# B&R Automation Studio project NAELD004C00R10L518F00 (part 18)

#### Act_OptP1030Save.st
```iecst
ACTION Act_OptP1030Save:

	CASE p_tyNtParamCurr.eProjMag OF
		LDMagDual, LDMagTriple:
			IF tyP1030MagSet.tyMagSet.tyBtnSave.bRtCompl = TRUE THEN
				IF usiSaveMagRcpStep = 0 THEN
					//Mask Table
					tyP1030MagSet.tyMagSet.tyTableRecipe.uiMaskRtStat				:= FALSE;
					tyP1030MagSet.tyMagSet.tyBtnDelete.uiMaskRtStat					:= FALSE;

					p_tyC0008MsgBox ACCESS ADR(tyP1030MagSet.tyMsgBoxSaveAsk);

					IF tyP1030MagSet.tyMsgBoxSaveAsk.tyBtnYes.bRtCompl = TRUE THEN
						tyP1030MagSet.tyMsgBoxSaveAsk.tyBtnYes.bRtCompl				:= FALSE;
						tyP1030MagSet.tyMsgBoxSaveAsk.tyBtnYes.bValue				:= FALSE;

						p_tyC0008MsgBox ACCESS ADR(tyP1030MagSet.tyMsgBoxHide);

						usiSaveMagRcpStep	:= 1;

					ELSIF tyP1030MagSet.tyMsgBoxSaveAsk.tyBtnNo.bRtCompl = TRUE THEN
						tyP1030MagSet.tyMsgBoxSaveAsk.tyBtnNo.bRtCompl				:= FALSE;
						tyP1030MagSet.tyMsgBoxSaveAsk.tyBtnNo.bValue				:= FALSE;

						p_tyC0008MsgBox ACCESS ADR(tyP1030MagSet.tyMsgBoxHide);

						usiSaveMagRcpStep	:= 99;

					END_IF

				ELSIF usiSaveMagRcpStep = 1 THEN
					tyMagRcpInfoIn.sRcpNm					:= tyP1030MagSet.tyMagSet.tyStringRecipeNm.sValue;
					tyMagRcpInfoIn.diSltToSltInUM			:= tyP1030MagSet.tyMagSet.tyNumSltToSltDist.diValue;
					tyMagRcpInfoIn.diTtlSlt					:= tyP1030MagSet.tyMagSet.tyNumMaxSlt.diValue;
					tyMagRcpInfoIn.diMag1Slt1PosInUM		:= tyP1030MagSet.tyMagSet.tyNumLifterMag1Slt1Pos.diValue;
					tyMagRcpInfoIn.diMag2Slt1PosInUM		:= tyP1030MagSet.tyMagSet.tyNumLifterMag2Slt1Pos.diValue;
					tyMagRcpInfoIn.diMag3Slt1PosInUM		:= tyP1030MagSet.tyMagSet.tyNumLifterMag3Slt1Pos.diValue;
					tyMagRcpInfoIn.diMag4Slt1PosInUM		:= tyP1030MagSet.tyMagSet.tyNumLifterMag4Slt1Pos.diValue;
					tyMagRcpInfoIn.diMag1TravPosInUM		:= tyP1030MagSet.tyMagSet.tyNumTravPosMag1.diValue;
					tyMagRcpInfoIn.diMag2TravPosInUM		:= tyP1030MagSet.tyMagSet.tyNumTravPosMag2.diValue;
					tyMagRcpInfoIn.diMag3TravPosInUM		:= tyP1030MagSet.tyMagSet.tyNumTravPosMag3.diValue;
					tyMagRcpInfoIn.diMag4TravPosInUM		:= tyP1030MagSet.tyMagSet.tyNumTravPosMag4.diValue;
					tyMagRcpInfoIn.usiMagModel				:= tyP1030MagSet.tyMagSet.tyDrpDnMagModel.usiValueIdx;
					tyMagRcpInfoIn.diMagMaxBrdWidth			:= tyP1030MagSet.tyMagSet.tyNumMagMaxBrdWidth.diValue;
					tyMagRcpInfoIn.bSafetyBarDisabled		:= tyP1030MagSet.tyMagSet.tyBtnSafetyBarDisabled.bValue;
					tyMagRcpInfoIn.bMagHeightChkEn			:= tyP1030MagSet.tyMagSet.tyBtnMagHeightChkEn.bValue;

					eMagRcpAct					:= MagRcpActAddEdit;

					IF p_eMagRcpStat = MagRcpActAddEdit AND p_eMagRcpStatus = Done THEN
						eMagRcpAct	:= MagRcpActIdle;

						IF p_bMagRcpNmEmpty = TRUE THEN
							usiSaveMagRcpStep		:= 2;
						ELSIF p_bMagRcpListFull = TRUE THEN
							usiSaveMagRcpStep		:= 3;
						ELSE
							bRefreshMagRcpTable	:= TRUE;
							bRefreshMagRcpDetail	:= TRUE;
							usiSaveMagRcpStep		:= 4;
						END_IF

					ELSIF p_eMagRcpStatus = Error THEN
						p_tyC0008MsgBox ACCESS ADR(tyP1030MagSet.tyMsgBoxSaveErr);

						IF tyP1030MagSet.tyMsgBoxSaveErr.tyBtnNo.bRtCompl = TRUE THEN
							tyP1030MagSet.tyMsgBoxSaveErr.tyBtnNo.bRtCompl 		:= FALSE;
							tyP1030MagSet.tyMsgBoxSaveErr.tyBtnNo.bValue 		:= FALSE;

							p_tyC0008MsgBox ACCESS ADR(tyP1030MagSet.tyMsgBoxHide);

							usiSaveMagRcpStep		:= 99;
						END_IF
					END_IF

				// Magazine Recipe Param Error
				ELSIF usiSaveMagRcpStep = 2 THEN
					p_tyC0008MsgBox ACCESS ADR(tyP1030MagSet.tyMsgBoxSaveNoNm);

					IF tyP1030MagSet.tyMsgBoxSaveNoNm.tyBtnNo.bRtCompl = TRUE THEN
						tyP1030MagSet.tyMsgBoxSaveNoNm.tyBtnNo.bRtCompl 			:= FALSE;
						tyP1030MagSet.tyMsgBoxSaveNoNm.tyBtnNo.bValue 				:= FALSE;

						p_tyC0008MsgBox ACCESS ADR(tyP1030MagSet.tyMsgBoxHide);

						usiSaveMagRcpStep		:= 99;
					END_IF

				// Magazine Recipe List Full
				ELSIF usiSaveMagRcpStep = 3 THEN
					p_tyC0008MsgBox ACCESS ADR(tyP1030MagSet.tyMsgBoxListFull);

					IF tyP1030MagSet.tyMsgBoxListFull.tyBtnNo.bRtCompl = TRUE THEN
						tyP1030MagSet.tyMsgBoxListFull.tyBtnNo.bRtCompl 				:= FALSE;
						tyP1030MagSet.tyMsgBoxListFull.tyBtnNo.bValue 					:= FALSE;

						p_tyC0008MsgBox ACCESS ADR(tyP1030MagSet.tyMsgBoxHide);

						usiSaveMagRcpStep		:= 99;
					END_IF

				ELSIF usiSaveMagRcpStep = 4 THEN
					IF tyMagRcpInfoIn.sRcpNm = p_tyMagRcpCurrRcp.sRcpNm THEN
						p_tyC0008MsgBox ACCESS ADR(tyP1030MagSet.tyMsgBoxReloadCurrRcp);

						IF tyP1030MagSet.tyMsgBoxReloadCurrRcp.tyBtnNo.bRtCompl = TRUE THEN
							tyP1030MagSet.tyMsgBoxReloadCurrRcp.tyBtnNo.bRtCompl 	:= FALSE;
							tyP1030MagSet.tyMsgBoxReloadCurrRcp.tyBtnNo.bValue 		:= FALSE;

							p_tyC0008MsgBox ACCESS ADR(tyP1030MagSet.tyMsgBoxHide);

							usiSaveMagRcpStep		:= 99;
						END_IF
					ELSE
						usiSaveMagRcpStep			:= 99;
					END_IF

				ELSIF usiSaveMagRcpStep = 99 THEN
					bRefreshMagRcpTable 			:= FALSE;

					//Unmask
					tyP1030MagSet.tyMagSet.tyTableRecipe.uiMaskRtStat	:= TRUE;
					tyP1030MagSet.tyMagSet.tyBtnDelete.uiMaskRtStat		:= TRUE;

					//Reset
					tyP1030MagSet.tyMagSet.tyBtnSave.bRtCompl	:= FALSE;
					tyP1030MagSet.tyMagSet.tyBtnSave.bValue		:= FALSE;

					usiSaveMagRcpStep	:= 0;

				END_IF

			END_IF

		LDMagQuadruple:
			IF tyP1030MagSet.tyMagSet.tyBtnSave.bRtCompl = TRUE THEN
				IF usiSaveMagRcpStep = 0 THEN
					//Mask Table
					tyP1030MagSet.tyMagSet.tyTableRecipe.uiMaskRtStat				:= FALSE;
					tyP1030MagSet.tyMagSet.tyBtnDelete.uiMaskRtStat					:= FALSE;

					p_tyC0008MsgBox ACCESS ADR(tyP1030MagSet.tyMsgBoxSaveAsk);

					IF tyP1030MagSet.tyMsgBoxSaveAsk.tyBtnYes.bRtCompl = TRUE THEN
						tyP1030MagSet.tyMsgBoxSaveAsk.tyBtnYes.bRtCompl				:= FALSE;
						tyP1030MagSet.tyMsgBoxSaveAsk.tyBtnYes.bValue				:= FALSE;

						p_tyC0008MsgBox ACCESS ADR(tyP1030MagSet.tyMsgBoxHide);

						usiSaveMagRcpStep	:= 1;

					ELSIF tyP1030MagSet.tyMsgBoxSaveAsk.tyBtnNo.bRtCompl = TRUE THEN
						tyP1030MagSet.tyMsgBoxSaveAsk.tyBtnNo.bRtCompl				:= FALSE;
						tyP1030MagSet.tyMsgBoxSaveAsk.tyBtnNo.bValue				:= FALSE;

						p_tyC0008MsgBox ACCESS ADR(tyP1030MagSet.tyMsgBoxHide);

						usiSaveMagRcpStep	:= 99;

					END_IF

				ELSIF usiSaveMagRcpStep = 1 THEN
					tyMagRcpInfoIn.sRcpNm					:= tyP1030MagSet.tyMagSet.tyStringRecipeNm.sValue;
					tyMagRcpInfoIn.diSltToSltInUM			:= tyP1030MagSet.tyMagSet.tyNumSltToSltDist.diValue;
					tyMagRcpInfoIn.diTtlSlt					:= tyP1030MagSet.tyMagSet.tyNumMaxSlt.diValue;
					tyMagRcpInfoIn.diMag1Slt1PosInUM		:= tyP1030MagSet.tyMagSet.tyNumLifterMag1Slt1Pos.diValue;
					tyMagRcpInfoIn.diMag2Slt1PosInUM		:= tyP1030MagSet.tyMagSet.tyNumLifterMag2Slt1Pos.diValue;
					tyMagRcpInfoIn.diMag3Slt1PosInUM		:= tyP1030MagSet.tyMagSet.tyNumLifterMag3Slt1Pos.diValue;
					tyMagRcpInfoIn.diMag4Slt1PosInUM		:= tyP1030MagSet.tyMagSet.tyNumLifterMag4Slt1Pos.diValue;
					tyMagRcpInfoIn.diMag1TravPosInUM		:= tyP1030MagSet.tyMagSet.tyNumTravPosMag1.diValue;
					tyMagRcpInfoIn.diMag2TravPosInUM		:= tyP1030MagSet.tyMagSet.tyNumTravPosMag2.diValue;
					tyMagRcpInfoIn.diMag3TravPosInUM		:= tyP1030MagSet.tyMagSet.tyNumTravPosMag3.diValue;
					tyMagRcpInfoIn.diMag4TravPosInUM		:= tyP1030MagSet.tyMagSet.tyNumTravPosMag4.diValue;
					tyMagRcpInfoIn.usiMagModel				:= tyP1030MagSet.tyMagSet.tyDrpDnMagModel.usiValueIdx;
					tyMagRcpInfoIn.diMagMaxBrdWidth			:= tyP1030MagSet.tyMagSet.tyNumMagMaxBrdWidth.diValue;
					tyMagRcpInfoIn.bSafetyBarDisabled		:= tyP1030MagSet.tyMagSet.tyBtnSafetyBarDisabled.bValue;

					tyMagRcpInfoIn1.sRcpNm					:= tyP1030MagSet.tyMagSet.tyStringRecipeNm.sValue;
					tyMagRcpInfoIn1.diSltToSltInUM			:= tyP1030MagSet.tyMagSet.tyNumSltToSltDist.diValue;
					tyMagRcpInfoIn1.diTtlSlt				:= tyP1030MagSet.tyMagSet.tyNumMaxSlt.diValue;
					tyMagRcpInfoIn1.diMag1Slt1PosInUM		:= tyP1030MagSet.tyMagSet.tyNumLifterMag1Slt1Pos.diValue;
					tyMagRcpInfoIn1.diMag2Slt1PosInUM		:= tyP1030MagSet.tyMagSet.tyNumLifterMag2Slt1Pos.diValue;
					tyMagRcpInfoIn1.diMag3Slt1PosInUM		:= tyP1030MagSet.tyMagSet.tyNumLifterMag3Slt1Pos.diValue;
					tyMagRcpInfoIn1.diMag4Slt1PosInUM		:= tyP1030MagSet.tyMagSet.tyNumLifterMag4Slt1Pos.diValue;
					tyMagRcpInfoIn1.diMag1TravPosInUM		:= tyP1030MagSet.tyMagSet.tyNumTravPosMag1.diValue;
					tyMagRcpInfoIn1.diMag2TravPosInUM		:= tyP1030MagSet.tyMagSet.tyNumTravPosMag2.diValue;
					tyMagRcpInfoIn1.diMag3TravPosInUM		:= tyP1030MagSet.tyMagSet.tyNumTravPosMag3.diValue;
					tyMagRcpInfoIn1.diMag4TravPosInUM		:= tyP1030MagSet.tyMagSet.tyNumTravPosMag4.diValue;
					tyMagRcpInfoIn1.usiMagModel				:= tyP1030MagSet.tyMagSet.tyDrpDnMagModel.usiValueIdx;
					tyMagRcpInfoIn1.diMagMaxBrdWidth		:= tyP1030MagSet.tyMagSet.tyNumMagMaxBrdWidth.diValue;
					tyMagRcpInfoIn1.bSafetyBarDisabled		:= tyP1030MagSet.tyMagSet.tyBtnSafetyBarDisabled.bValue;
					tyMagRcpInfoIn1.bMagHeightChkEn			:= tyP1030MagSet.tyMagSet.tyBtnMagHeightChkEn.bValue;

					eMagRcpAct					:= MagRcpActAddEdit;
					eMagRcpAct1					:= MagRcpActAddEdit;

					IF (p_eMagRcpStat = MagRcpActAddEdit AND p_eMagRcpStatus = Done)
						AND (p_eMagRcpStat1 = MagRcpActAddEdit AND p_eMagRcpStatus1 = Done)
						THEN
							eMagRcpAct	:= MagRcpActIdle;
							eMagRcpAct1	:= MagRcpActIdle;

						IF p_bMagRcpNmEmpty = TRUE OR p_bMagRcpNmEmpty1 = TRUE THEN
							usiSaveMagRcpStep		:= 2;
						ELSIF p_bMagRcpListFull = TRUE OR p_bMagRcpListFull1 = TRUE THEN
							usiSaveMagRcpStep		:= 3;
						ELSE
							bRefreshMagRcpTable	:= TRUE;
							bRefreshMagRcpDetail	:= TRUE;
							usiSaveMagRcpStep		:= 4;
						END_IF

					ELSIF p_eMagRcpStatus = Error OR p_eMagRcpStatus1 = Error THEN
						p_tyC0008MsgBox ACCESS ADR(tyP1030MagSet.tyMsgBoxSaveErr);

						IF tyP1030MagSet.tyMsgBoxSaveErr.tyBtnNo.bRtCompl = TRUE THEN
							tyP1030MagSet.tyMsgBoxSaveErr.tyBtnNo.bRtCompl 		:= FALSE;
							tyP1030MagSet.tyMsgBoxSaveErr.tyBtnNo.bValue 		:= FALSE;

							p_tyC0008MsgBox ACCESS ADR(tyP1030MagSet.tyMsgBoxHide);

							usiSaveMagRcpStep		:= 99;
						END_IF
					END_IF

					// Magazine Recipe Param Error
				ELSIF usiSaveMagRcpStep = 2 THEN
					p_tyC0008MsgBox ACCESS ADR(tyP1030MagSet.tyMsgBoxSaveNoNm);

					IF tyP1030MagSet.tyMsgBoxSaveNoNm.tyBtnNo.bRtCompl = TRUE THEN
						tyP1030MagSet.tyMsgBoxSaveNoNm.tyBtnNo.bRtCompl 			:= FALSE;
						tyP1030MagSet.tyMsgBoxSaveNoNm.tyBtnNo.bValue 				:= FALSE;

						p_tyC0008MsgBox ACCESS ADR(tyP1030MagSet.tyMsgBoxHide);

						usiSaveMagRcpStep		:= 99;
					END_IF

					// Magazine Recipe List Full
				ELSIF usiSaveMagRcpStep = 3 THEN
					p_tyC0008MsgBox ACCESS ADR(tyP1030MagSet.tyMsgBoxListFull);

					IF tyP1030MagSet.tyMsgBoxListFull.tyBtnNo.bRtCompl = TRUE THEN
						tyP1030MagSet.tyMsgBoxListFull.tyBtnNo.bRtCompl 				:= FALSE;
						tyP1030MagSet.tyMsgBoxListFull.tyBtnNo.bValue 					:= FALSE;

						p_tyC0008MsgBox ACCESS ADR(tyP1030MagSet.tyMsgBoxHide);

						usiSaveMagRcpStep		:= 99;
					END_IF

				ELSIF usiSaveMagRcpStep = 4 THEN
					IF tyMagRcpInfoIn.sRcpNm = p_tyMagRcpCurrRcp.sRcpNm OR tyMagRcpInfoIn1.sRcpNm = p_tyMagRcpCurrRcp1.sRcpNm THEN
						p_tyC0008MsgBox ACCESS ADR(tyP1030MagSet.tyMsgBoxReloadCurrRcp);

						IF tyP1030MagSet.tyMsgBoxReloadCurrRcp.tyBtnNo.bRtCompl = TRUE THEN
							tyP1030MagSet.tyMsgBoxReloadCurrRcp.tyBtnNo.bRtCompl 	:= FALSE;
							tyP1030MagSet.tyMsgBoxReloadCurrRcp.tyBtnNo.bValue 		:= FALSE;

							p_tyC0008MsgBox ACCESS ADR(tyP1030MagSet.tyMsgBoxHide);

							usiSaveMagRcpStep		:= 99;
						END_IF
					ELSE
						usiSaveMagRcpStep			:= 99;
					END_IF

				ELSIF usiSaveMagRcpStep = 99 THEN
					bRefreshMagRcpTable 			:= FALSE;

					//Unmask
					tyP1030MagSet.tyMagSet.tyTableRecipe.uiMaskRtStat	:= TRUE;
					tyP1030MagSet.tyMagSet.tyBtnDelete.uiMaskRtStat		:= TRUE;

					//Reset
					tyP1030MagSet.tyMagSet.tyBtnSave.bRtCompl	:= FALSE;
					tyP1030MagSet.tyMagSet.tyBtnSave.bValue		:= FALSE;

					usiSaveMagRcpStep	:= 0;

				END_IF

			END_IF
	END_CASE

END_ACTION
```

#### Act_OptP1030Teach.st
```iecst
ACTION Act_OptP1030Teach:

	IF tyP1030MagSet.tyMagSet.tyBtnLifterMag1Slt1Pos.bRtCompl = TRUE THEN
		tyP1030MagSet.tyMagSet.tyBtnLifterMag1Slt1Pos.bRtCompl	:= FALSE;
		tyP1030MagSet.tyMagSet.tyBtnLifterMag1Slt1Pos.bValue	:= FALSE;

		bTeachLifterMag1Slt1Pos	:= TRUE;
		eChgPage				:= UIP1031MagSetTeach;

	ELSIF tyP1030MagSet.tyMagSet.tyBtnLifterMag2Slt1Pos.bRtCompl = TRUE THEN
		tyP1030MagSet.tyMagSet.tyBtnLifterMag2Slt1Pos.bRtCompl	:= FALSE;
		tyP1030MagSet.tyMagSet.tyBtnLifterMag2Slt1Pos.bValue	:= FALSE;

		bTeachLifterMag2Slt1Pos	:= TRUE;
		eChgPage				:= UIP1031MagSetTeach;

	ELSIF tyP1030MagSet.tyMagSet.tyBtnLifterMag3Slt1Pos.bRtCompl = TRUE THEN
		tyP1030MagSet.tyMagSet.tyBtnLifterMag3Slt1Pos.bRtCompl	:= FALSE;
		tyP1030MagSet.tyMagSet.tyBtnLifterMag3Slt1Pos.bValue	:= FALSE;

		bTeachLifterMag3Slt1Pos	:= TRUE;
		eChgPage				:= UIP1031MagSetTeach;

	ELSIF tyP1030MagSet.tyMagSet.tyBtnLifterMag4Slt1Pos.bRtCompl = TRUE THEN
		tyP1030MagSet.tyMagSet.tyBtnLifterMag4Slt1Pos.bRtCompl	:= FALSE;
		tyP1030MagSet.tyMagSet.tyBtnLifterMag4Slt1Pos.bValue	:= FALSE;

		bTeachLifterMag4Slt1Pos	:= TRUE;
		eChgPage				:= UIP1031MagSetTeach;

	ELSIF tyP1030MagSet.tyMagSet.tyBtnTravPosMag1.bRtCompl = TRUE THEN
		tyP1030MagSet.tyMagSet.tyBtnTravPosMag1.bRtCompl	:= FALSE;
		tyP1030MagSet.tyMagSet.tyBtnTravPosMag1.bValue		:= FALSE;

		bTeachTravPosMag1	:= TRUE;
		eChgPage			:= UIP1031MagSetTeach;

	ELSIF tyP1030MagSet.tyMagSet.tyBtnTravPosMag2.bRtCompl = TRUE THEN
		tyP1030MagSet.tyMagSet.tyBtnTravPosMag2.bRtCompl	:= FALSE;
		tyP1030MagSet.tyMagSet.tyBtnTravPosMag2.bValue		:= FALSE;

		bTeachTravPosMag2	:= TRUE;
		eChgPage			:= UIP1031MagSetTeach;

	ELSIF tyP1030MagSet.tyMagSet.tyBtnTravPosMag3.bRtCompl = TRUE THEN
		tyP1030MagSet.tyMagSet.tyBtnTravPosMag3.bRtCompl	:= FALSE;
		tyP1030MagSet.tyMagSet.tyBtnTravPosMag3.bValue		:= FALSE;

		bTeachTravPosMag3	:= TRUE;
		eChgPage			:= UIP1031MagSetTeach;

	ELSIF tyP1030MagSet.tyMagSet.tyBtnTravPosMag4.bRtCompl = TRUE THEN
		tyP1030MagSet.tyMagSet.tyBtnTravPosMag4.bRtCompl	:= FALSE;
		tyP1030MagSet.tyMagSet.tyBtnTravPosMag4.bValue		:= FALSE;

		bTeachTravPosMag4	:= TRUE;
		eChgPage			:= UIP1031MagSetTeach;

	END_IF

END_ACTION
```

#### Act_EntP1031Disp.st
```iecst
ACTION Act_EntP1031Disp:

	//Access Address
	p_tyC0002FullMask ACCESS ADR(tyP1031MagSetTeach.tyFullMaskHide);

	p_tyC0004Navi ACCESS ADR(tyP1031MagSetTeach.tyNaviBack);

	p_tyC0005Main ACCESS ADR(tyCommon.tyMain);

	p_tyC0007Notif ACCESS ADR(tyCommon.tyNotif);

	p_tyC0008MsgBox ACCESS ADR(tyP1031MagSetTeach.tyMsgBoxHide);

	p_tyC0009Info ACCESS ADR(tyCommon.tyInfo);

	p_tyP1031InOutletShutterFB ACCESS ADR(tyP1031MagSetTeach.tyInOutletShutterFB);

//	bTeachServo		:= TRUE;

	IF bTeachLifterMag1Slt1Pos = TRUE THEN
		tyP1031MagSetTeach.tyTeachLifterMag1Slt1Pos.tyNumNewSlt.diValue := 1;
		tyP1031MagSetTeach.tyTeachLifterMag1Slt1Pos.tyNumNewSlt.diValueMin := 1;
		tyP1031MagSetTeach.tyTeachLifterMag1Slt1Pos.tyNumNewSlt.diValueMax := tyP1030MagSet.tyMagSet.tyNumMaxSlt.diValue;

		p_tyP1031MagSetTeach ACCESS ADR(tyP1031MagSetTeach.tyTeachLifterMag1Slt1Pos);
		p_tyC0001MotionStd ACCESS ADR(tyP1031MagSetTeach.tyMotionStdLifter);

	ELSIF bTeachLifterMag2Slt1Pos = TRUE THEN
		tyP1031MagSetTeach.tyTeachLifterMag2Slt1Pos.tyNumNewSlt.diValue := 1;
		tyP1031MagSetTeach.tyTeachLifterMag2Slt1Pos.tyNumNewSlt.diValueMin := 1;
		tyP1031MagSetTeach.tyTeachLifterMag2Slt1Pos.tyNumNewSlt.diValueMax := tyP1030MagSet.tyMagSet.tyNumMaxSlt.diValue;

		p_tyP1031MagSetTeach ACCESS ADR(tyP1031MagSetTeach.tyTeachLifterMag2Slt1Pos);
		p_tyC0001MotionStd ACCESS ADR(tyP1031MagSetTeach.tyMotionStdLifter);

	ELSIF bTeachLifterMag3Slt1Pos = TRUE THEN
		tyP1031MagSetTeach.tyTeachLifterMag3Slt1Pos.tyNumNewSlt.diValue := 1;
		tyP1031MagSetTeach.tyTeachLifterMag3Slt1Pos.tyNumNewSlt.diValueMin := 1;
		tyP1031MagSetTeach.tyTeachLifterMag3Slt1Pos.tyNumNewSlt.diValueMax := tyP1030MagSet.tyMagSet.tyNumMaxSlt.diValue;

		p_tyP1031MagSetTeach ACCESS ADR(tyP1031MagSetTeach.tyTeachLifterMag3Slt1Pos);
		p_tyC0001MotionStd ACCESS ADR(tyP1031MagSetTeach.tyMotionStdLifter);

	ELSIF bTeachLifterMag4Slt1Pos = TRUE THEN
		tyP1031MagSetTeach.tyTeachLifterMag4Slt1Pos.tyNumNewSlt.diValue := 1;
		tyP1031MagSetTeach.tyTeachLifterMag4Slt1Pos.tyNumNewSlt.diValueMin := 1;
		tyP1031MagSetTeach.tyTeachLifterMag4Slt1Pos.tyNumNewSlt.diValueMax := tyP1030MagSet.tyMagSet.tyNumMaxSlt.diValue;

		p_tyP1031MagSetTeach ACCESS ADR(tyP1031MagSetTeach.tyTeachLifterMag4Slt1Pos);
		p_tyC0001MotionStd ACCESS ADR(tyP1031MagSetTeach.tyMotionStdLifter);

	ELSIF bTeachTravPosMag1 = TRUE THEN
		tyP1031MagSetTeach.tyTeachTravPosMag1.tyNumNewSlt.uiRtStat.0 := TRUE;

		p_tyP1031MagSetTeach ACCESS ADR(tyP1031MagSetTeach.tyTeachTravPosMag1);
		p_tyC0001MotionStd ACCESS ADR(tyP1031MagSetTeach.tyMotionStdTrav);

	ELSIF bTeachTravPosMag2 = TRUE THEN
		tyP1031MagSetTeach.tyTeachTravPosMag2.tyNumNewSlt.uiRtStat.0 := TRUE;

		p_tyP1031MagSetTeach ACCESS ADR(tyP1031MagSetTeach.tyTeachTravPosMag2);
		p_tyC0001MotionStd ACCESS ADR(tyP1031MagSetTeach.tyMotionStdTrav);

	ELSIF bTeachTravPosMag3 = TRUE THEN
		tyP1031MagSetTeach.tyTeachTravPosMag3.tyNumNewSlt.uiRtStat.0 := TRUE;

		p_tyP1031MagSetTeach ACCESS ADR(tyP1031MagSetTeach.tyTeachTravPosMag3);
		p_tyC0001MotionStd ACCESS ADR(tyP1031MagSetTeach.tyMotionStdTrav);

	ELSIF bTeachTravPosMag4 = TRUE THEN
		tyP1031MagSetTeach.tyTeachTravPosMag4.tyNumNewSlt.uiRtStat.0 := TRUE;

		p_tyP1031MagSetTeach ACCESS ADR(tyP1031MagSetTeach.tyTeachTravPosMag4);
		p_tyC0001MotionStd ACCESS ADR(tyP1031MagSetTeach.tyMotionStdTrav);

	END_IF

	//Display
	//Traverser
	tyP1031MagSetTeach.tyMotionStdTrav.tyBtnPwr.bValue	:= p_bTravPwrOn;

	//Lifter
	tyP1031MagSetTeach.tyMotionStdLifter.tyBtnPwr.bValue	:= p_bLifterBtmPwrOn;

END_ACTION
```

#### Act_ExitP1031.st
```iecst
ACTION Act_ExitP1031:

	usiChgPage	:= 1;

	//Manual Deactivated
	bManualMod	:= FALSE;

	//Reset UI
	bJogSlow				:= FALSE;
	bJogFast				:= FALSE;
	fbJogSlowToFastDlyTm.IN	:= FALSE;
	bTeachServo				:= FALSE;

	fbLmtRstTm(IN := FALSE);
	//bypass curtain sensor
	bBypCurtainSen := FALSE;
	bBypCurtainPBLED := FALSE;
	tyP1031MagSetTeach.tyTeachTravPosMag1.tyBtn4.bValue				:= FALSE;
	tyP1031MagSetTeach.tyTeachTravPosMag2.tyBtn4.bValue				:= FALSE;
	tyP1031MagSetTeach.tyTeachTravPosMag3.tyBtn4.bValue				:= FALSE;
	tyP1031MagSetTeach.tyTeachLifterMag1Slt1Pos.tyBtn4.bValue				:= FALSE;
	tyP1031MagSetTeach.tyTeachLifterMag2Slt1Pos.tyBtn4.bValue				:= FALSE;
	tyP1031MagSetTeach.tyTeachLifterMag3Slt1Pos.tyBtn4.bValue				:= FALSE;

	//Traverser
	tyP1031MagSetTeach.tyMotionStdTrav.tyBtnPwr.bRtCompl			:= FALSE;
	tyP1031MagSetTeach.tyMotionStdTrav.tyBtnStop.bRtCompl			:= FALSE;
	tyP1031MagSetTeach.tyMotionStdTrav.tyBtnOrigin.bRtCompl			:= FALSE;
	tyP1031MagSetTeach.tyMotionStdTrav.tyBtnRst.bRtCompl			:= FALSE;
	tyP1031MagSetTeach.tyMotionStdTrav.tyBtnMovAbs.bRtCompl			:= FALSE;
	tyP1031MagSetTeach.tyMotionStdTrav.tyBtnMovRel.bRtCompl			:= FALSE;
	tyP1031MagSetTeach.tyMotionStdTrav.tyBtnJogFront.bRtCompl		:= FALSE;
	tyP1031MagSetTeach.tyMotionStdTrav.tyBtnJogRear.bRtCompl		:= FALSE;

	tyP1031MagSetTeach.tyTeachTravPosMag1.tyBtn2.bRtCompl			:= FALSE;
	tyP1031MagSetTeach.tyTeachTravPosMag2.tyBtn2.bRtCompl			:= FALSE;
	tyP1031MagSetTeach.tyTeachTravPosMag3.tyBtn2.bRtCompl			:= FALSE;

	tyP1031MagSetTeach.tyMotionStdTrav.tyBtnPwr.bValue				:= FALSE;
	tyP1031MagSetTeach.tyMotionStdTrav.tyBtnStop.bValue				:= TRUE;
	tyP1031MagSetTeach.tyMotionStdTrav.tyBtnOrigin.bValue			:= FALSE;
	tyP1031MagSetTeach.tyMotionStdTrav.tyBtnRst.bValue				:= FALSE;
	tyP1031MagSetTeach.tyMotionStdTrav.tyBtnMovAbs.bValue			:= FALSE;
	tyP1031MagSetTeach.tyMotionStdTrav.tyBtnMovRel.bValue			:= FALSE;
	tyP1031MagSetTeach.tyMotionStdTrav.tyBtnJogFront.bValue			:= FALSE;
	tyP1031MagSetTeach.tyMotionStdTrav.tyBtnJogRear.bValue			:= FALSE;

	tyP1031MagSetTeach.tyTeachTravPosMag1.tyBtn2.bValue				:= FALSE;
	tyP1031MagSetTeach.tyTeachTravPosMag2.tyBtn2.bValue				:= FALSE;
	tyP1031MagSetTeach.tyTeachTravPosMag3.tyBtn2.bValue				:= FALSE;

	tyP1031MagSetTeach.tyMotionStdTrav.tyBtnPwr.bRtLk				:= FALSE;
	tyP1031MagSetTeach.tyMotionStdTrav.tyBtnStop.bRtLk				:= TRUE;
	tyP1031MagSetTeach.tyMotionStdTrav.tyBtnOrigin.bRtLk			:= FALSE;
	tyP1031MagSetTeach.tyMotionStdTrav.tyBtnRst.bRtLk				:= FALSE;
	tyP1031MagSetTeach.tyMotionStdTrav.tyBtnMovAbs.bRtLk			:= FALSE;
	tyP1031MagSetTeach.tyMotionStdTrav.tyBtnMovRel.bRtLk			:= FALSE;
	tyP1031MagSetTeach.tyMotionStdTrav.tyBtnJogFront.bRtLk			:= FALSE;
	tyP1031MagSetTeach.tyMotionStdTrav.tyBtnJogRear.bRtLk			:= FALSE;

	tyP1031MagSetTeach.tyTeachTravPosMag1.tyBtn2.bRtLk				:= FALSE;
	tyP1031MagSetTeach.tyTeachTravPosMag2.tyBtn2.bRtLk				:= FALSE;
	tyP1031MagSetTeach.tyTeachTravPosMag3.tyBtn2.bRtLk				:= FALSE;

	tyP1031MagSetTeach.tyMotionStdTrav.tyBtnPwr.uiMaskRtStat		:= TRUE;
	tyP1031MagSetTeach.tyMotionStdTrav.tyBtnOrigin.uiMaskRtStat		:= FALSE;
	tyP1031MagSetTeach.tyMotionStdTrav.tyBtnRst.uiMaskRtStat		:= TRUE;
	tyP1031MagSetTeach.tyMotionStdTrav.tyBtnMovAbs.uiMaskRtStat		:= FALSE;
	tyP1031MagSetTeach.tyMotionStdTrav.tyBtnMovRel.uiMaskRtStat		:= FALSE;
	tyP1031MagSetTeach.tyMotionStdTrav.tyBtnJogFront.uiMaskRtStat	:= FALSE;
	tyP1031MagSetTeach.tyMotionStdTrav.tyBtnJogRear.uiMaskRtStat	:= FALSE;

	tyP1031MagSetTeach.tyTeachTravPosMag1.tyBtn2.uiMaskRtStat		:= FALSE;
	tyP1031MagSetTeach.tyTeachTravPosMag2.tyBtn2.uiMaskRtStat		:= FALSE;
	tyP1031MagSetTeach.tyTeachTravPosMag3.tyBtn2.uiMaskRtStat		:= FALSE;

	//Lifter
	tyP1031MagSetTeach.tyMotionStdLifter.tyBtnPwr.bRtCompl			:= FALSE;
	tyP1031MagSetTeach.tyMotionStdLifter.tyBtnStop.bRtCompl			:= FALSE;
	tyP1031MagSetTeach.tyMotionStdLifter.tyBtnOrigin.bRtCompl		:= FALSE;
	tyP1031MagSetTeach.tyMotionStdLifter.tyBtnRst.bRtCompl			:= FALSE;
	tyP1031MagSetTeach.tyMotionStdLifter.tyBtnMovAbs.bRtCompl		:= FALSE;
	tyP1031MagSetTeach.tyMotionStdLifter.tyBtnMovRel.bRtCompl		:= FALSE;
	tyP1031MagSetTeach.tyMotionStdLifter.tyBtnJogUp.bRtCompl		:= FALSE;
	tyP1031MagSetTeach.tyMotionStdLifter.tyBtnJogDown.bRtCompl		:= FALSE;

	tyP1031MagSetTeach.tyTeachLifterMag1Slt1Pos.tyBtn2.bRtCompl		:= FALSE;
	tyP1031MagSetTeach.tyTeachLifterMag2Slt1Pos.tyBtn2.bRtCompl		:= FALSE;
	tyP1031MagSetTeach.tyTeachLifterMag3Slt1Pos.tyBtn2.bRtCompl		:= FALSE;

	tyP1031MagSetTeach.tyMotionStdLifter.tyBtnPwr.bValue			:= FALSE;
	tyP1031MagSetTeach.tyMotionStdLifter.tyBtnStop.bValue			:= TRUE;
	tyP1031MagSetTeach.tyMotionStdLifter.tyBtnOrigin.bValue			:= FALSE;
	tyP1031MagSetTeach.tyMotionStdLifter.tyBtnRst.bValue			:= FALSE;
	tyP1031MagSetTeach.tyMotionStdLifter.tyBtnMovAbs.bValue			:= FALSE;
	tyP1031MagSetTeach.tyMotionStdLifter.tyBtnMovRel.bValue			:= FALSE;
	tyP1031MagSetTeach.tyMotionStdLifter.tyBtnJogUp.bValue			:= FALSE;
	tyP1031MagSetTeach.tyMotionStdLifter.tyBtnJogDown.bValue		:= FALSE;

	tyP1031MagSetTeach.tyTeachLifterMag1Slt1Pos.tyBtn2.bValue		:= FALSE;
	tyP1031MagSetTeach.tyTeachLifterMag2Slt1Pos.tyBtn2.bValue		:= FALSE;
	tyP1031MagSetTeach.tyTeachLifterMag3Slt1Pos.tyBtn2.bValue		:= FALSE;

	tyP1031MagSetTeach.tyMotionStdLifter.tyBtnPwr.bRtLk				:= FALSE;
	tyP1031MagSetTeach.tyMotionStdLifter.tyBtnStop.bRtLk			:= TRUE;
	tyP1031MagSetTeach.tyMotionStdLifter.tyBtnOrigin.bRtLk			:= FALSE;
	tyP1031MagSetTeach.tyMotionStdLifter.tyBtnRst.bRtLk				:= FALSE;
	tyP1031MagSetTeach.tyMotionStdLifter.tyBtnMovAbs.bRtLk			:= FALSE;
	tyP1031MagSetTeach.tyMotionStdLifter.tyBtnMovRel.bRtLk			:= FALSE;
	tyP1031MagSetTeach.tyMotionStdLifter.tyBtnJogUp.bRtLk			:= FALSE;
	tyP1031MagSetTeach.tyMotionStdLifter.tyBtnJogDown.bRtLk			:= FALSE;

	tyP1031MagSetTeach.tyTeachLifterMag1Slt1Pos.tyBtn2.bRtLk		:= FALSE;
	tyP1031MagSetTeach.tyTeachLifterMag2Slt1Pos.tyBtn2.bRtLk		:= FALSE;
	tyP1031MagSetTeach.tyTeachLifterMag3Slt1Pos.tyBtn2.bRtLk		:= FALSE;

	tyP1031MagSetTeach.tyMotionStdLifter.tyBtnPwr.uiMaskRtStat		:= TRUE;
	tyP1031MagSetTeach.tyMotionStdLifter.tyBtnOrigin.uiMaskRtStat	:= FALSE;
	tyP1031MagSetTeach.tyMotionStdLifter.tyBtnRst.uiMaskRtStat		:= TRUE;
	tyP1031MagSetTeach.tyMotionStdLifter.tyBtnMovAbs.uiMaskRtStat	:= FALSE;
	tyP1031MagSetTeach.tyMotionStdLifter.tyBtnMovRel.uiMaskRtStat	:= FALSE;
	tyP1031MagSetTeach.tyMotionStdLifter.tyBtnJogUp.uiMaskRtStat	:= FALSE;
	tyP1031MagSetTeach.tyMotionStdLifter.tyBtnJogDown.uiMaskRtStat	:= FALSE;

	tyP1031MagSetTeach.tyTeachLifterMag1Slt1Pos.tyBtn2.uiMaskRtStat	:= FALSE;
	tyP1031MagSetTeach.tyTeachLifterMag2Slt1Pos.tyBtn2.uiMaskRtStat	:= FALSE;
	tyP1031MagSetTeach.tyTeachLifterMag3Slt1Pos.tyBtn2.uiMaskRtStat	:= FALSE;

END_ACTION
```

#### Act_OptP1031FullMask.st
```iecst
ACTION Act_OptP1031FullMask:

	IF eCurrPage = UIP1031MagSetTeach THEN

		IF p_tyDI.bEStopSig = FALSE THEN
			p_tyC0002FullMask ACCESS ADR(tyP1031MagSetTeach.tyFullMaskEStop);

		ELSIF p_tyDI.bCoverSWSig = FALSE THEN
			p_tyC0002FullMask ACCESS ADR(tyP1031MagSetTeach.tyFullMaskCWSig);

		ELSIF p_tyDI.bSafetyRlySig = FALSE THEN
			p_tyC0002FullMask ACCESS ADR(tyP1031MagSetTeach.tyFullMaskSafetyRly);

		ELSIF p_tyDI.bLifterSafetyLmtSW1 = FALSE OR p_tyDI.bLifterSafetyLmtSW2 = FALSE THEN
			p_tyC0002FullMask ACCESS ADR(tyP1031MagSetTeach.tyFullMaskSafetyLmtSW);

		ELSIF p_tyDI.bLifterTimingBeltSen = FALSE THEN
			p_tyC0002FullMask ACCESS ADR(tyP1031MagSetTeach.tyFullMaskTimingBelt);

		ELSE
			p_tyC0002FullMask ACCESS ADR(tyP1031MagSetTeach.tyFullMaskHide);

		END_IF

	END_IF

END_ACTION
```

#### Act_OptP1031TravTeach.st
```iecst
ACTION Act_OptP1031TravTeach:

	IF tyP1031MagSetTeach.tyTeachTravPosMag1.tyBtn1.bRtCompl = TRUE THEN

		p_tyC0008MsgBox ACCESS ADR(tyP1031MagSetTeach.tyMsgBoxUpdtTravPosMag1);

		IF tyP1031MagSetTeach.tyMsgBoxUpdtTravPosMag1.tyBtnNo.bRtCompl THEN
			tyP1031MagSetTeach.tyMsgBoxUpdtTravPosMag1.tyBtnNo.bRtCompl := FALSE;
			tyP1031MagSetTeach.tyMsgBoxUpdtTravPosMag1.tyBtnNo.bValue 	:= FALSE;

			p_tyC0008MsgBox ACCESS ADR(tyP1031MagSetTeach.tyMsgBoxHide);

			//Write Actual Position To Magazine Setting.
			tyP1030MagSet.tyMagSet.tyNumTravPosMag1.diValue 	:= p_diTravActualPos;
			tyP1030MagSet.tyMagSet.tyNumTravPosMag1.bRtCompl	:= TRUE;

			//Back To Magazine Settings
			eChgPage	:= UIP1030MagSet;

			fUIInRtStatHide(ADR(tyP1030MagSet.tyMagSet.tyBtnSave.uiMaskRtStat));

			tyP1031MagSetTeach.tyTeachTravPosMag1.tyBtn1.bRtCompl	:= FALSE;
			tyP1031MagSetTeach.tyTeachTravPosMag1.tyBtn1.bValue		:= FALSE;

		END_IF

	ELSIF tyP1031MagSetTeach.tyTeachTravPosMag2.tyBtn1.bRtCompl = TRUE THEN

		p_tyC0008MsgBox ACCESS ADR(tyP1031MagSetTeach.tyMsgBoxUpdtTravPosMag2);

		IF tyP1031MagSetTeach.tyMsgBoxUpdtTravPosMag2.tyBtnNo.bRtCompl THEN
			tyP1031MagSetTeach.tyMsgBoxUpdtTravPosMag2.tyBtnNo.bRtCompl := FALSE;
			tyP1031MagSetTeach.tyMsgBoxUpdtTravPosMag2.tyBtnNo.bValue 	:= FALSE;

			p_tyC0008MsgBox ACCESS ADR(tyP1031MagSetTeach.tyMsgBoxHide);

			//Write Actual Position To Magazine Setting.
			tyP1030MagSet.tyMagSet.tyNumTravPosMag2.diValue		:= p_diTravActualPos;
			tyP1030MagSet.tyMagSet.tyNumTravPosMag2.bRtCompl	:= TRUE;

			//Back To Magazine Settings
			eChgPage	:= UIP1030MagSet;

			fUIInRtStatHide(ADR(tyP1030MagSet.tyMagSet.tyBtnSave.uiMaskRtStat));

			tyP1031MagSetTeach.tyTeachTravPosMag2.tyBtn1.bRtCompl	:= FALSE;
			tyP1031MagSetTeach.tyTeachTravPosMag2.tyBtn1.bValue		:= FALSE;

		END_IF

	ELSIF tyP1031MagSetTeach.tyTeachTravPosMag3.tyBtn1.bRtCompl = TRUE THEN

		p_tyC0008MsgBox ACCESS ADR(tyP1031MagSetTeach.tyMsgBoxUpdtTravPosMag3);

		IF tyP1031MagSetTeach.tyMsgBoxUpdtTravPosMag3.tyBtnNo.bRtCompl THEN
			tyP1031MagSetTeach.tyMsgBoxUpdtTravPosMag3.tyBtnNo.bRtCompl := FALSE;
			tyP1031MagSetTeach.tyMsgBoxUpdtTravPosMag3.tyBtnNo.bValue 	:= FALSE;

			p_tyC0008MsgBox ACCESS ADR(tyP1031MagSetTeach.tyMsgBoxHide);

			//Write Actual Position To Magazine Setting.
			tyP1030MagSet.tyMagSet.tyNumTravPosMag3.diValue 	:= p_diTravActualPos;
			tyP1030MagSet.tyMagSet.tyNumTravPosMag3.bRtCompl	:= TRUE;

			//Back To Magazine Settings
			eChgPage	:= UIP1030MagSet;

			fUIInRtStatHide(ADR(tyP1030MagSet.tyMagSet.tyBtnSave.uiMaskRtStat));

			tyP1031MagSetTeach.tyTeachTravPosMag3.tyBtn1.bRtCompl	:= FALSE;
			tyP1031MagSetTeach.tyTeachTravPosMag3.tyBtn1.bValue		:= FALSE;

		END_IF

	ELSIF tyP1031MagSetTeach.tyTeachTravPosMag4.tyBtn1.bRtCompl = TRUE THEN

		p_tyC0008MsgBox ACCESS ADR(tyP1031MagSetTeach.tyMsgBoxUpdtTravPosMag4);

		IF tyP1031MagSetTeach.tyMsgBoxUpdtTravPosMag4.tyBtnNo.bRtCompl THEN
			tyP1031MagSetTeach.tyMsgBoxUpdtTravPosMag4.tyBtnNo.bRtCompl := FALSE;
			tyP1031MagSetTeach.tyMsgBoxUpdtTravPosMag4.tyBtnNo.bValue 	:= FALSE;

			p_tyC0008MsgBox ACCESS ADR(tyP1031MagSetTeach.tyMsgBoxHide);

			//Write Actual Position To Magazine Setting.
			tyP1030MagSet.tyMagSet.tyNumTravPosMag4.diValue 	:= p_diTravActualPos;
			tyP1030MagSet.tyMagSet.tyNumTravPosMag4.bRtCompl	:= TRUE;

			//Back To Magazine Settings
			eChgPage	:= UIP1030MagSet;

			fUIInRtStatHide(ADR(tyP1030MagSet.tyMagSet.tyBtnSave.uiMaskRtStat));

			tyP1031MagSetTeach.tyTeachTravPosMag4.tyBtn1.bRtCompl	:= FALSE;
			tyP1031MagSetTeach.tyTeachTravPosMag4.tyBtn1.bValue		:= FALSE;

		END_IF
	END_IF

END_ACTION
```

#### Act_OptP1031TravFBCtrl.st
```iecst
ACTION Act_OptP1031TravFBCtrl:

	fbJogSlowToFastDlyTm.PT			:= T#2s;
	fbJogSlowToFastDlyTm;
	fbLmtRstTm;

//	IF EDGEPOS((p_udiTravAxisErrID = 21570 OR p_udiTravAxisErrID = 21571)
	IF EDGEPOS((p_bTravFwdLmtSen OR p_bTravRevLmtSen OR p_udiTravAxisErrID = 21570 OR p_udiTravAxisErrID = 21571)
		AND tyP1031MagSetTeach.tyMotionStdTrav.tyBtnJogRear.bValue = FALSE
		AND tyP1031MagSetTeach.tyMotionStdTrav.tyBtnJogFront.bValue = FALSE) THEN
		fbLmtRstTm.IN				:= TRUE;
	END_IF

	IF fbLmtRstTm.Q = TRUE THEN
		tyP1031MagSetTeach.tyMotionStdTrav.tyBtnRst.bRtCompl		:= TRUE;
	END_IF

	IF (tyP1031MagSetTeach.tyMotionStdTrav.tyBtnJogFront.bValue = FALSE AND tyP1031MagSetTeach.tyMotionStdTrav.tyBtnJogRear.bValue = FALSE) AND (p_bTravJogging = TRUE) THEN
		bJogStopTrav	:= TRUE;
	END_IF

	IF tyP1031MagSetTeach.tyMotionStdTrav.tyBtnStop.bRtCompl = TRUE THEN
		eTravAct		:= TravActStop;

		IF p_eTravStat = TravActStop AND p_eTravStatus = Done THEN
			eTravAct	:= TravActIdle;

			tyP1031MagSetTeach.tyMotionStdTrav.tyBtnStop.bRtCompl		:= FALSE;
			tyP1031MagSetTeach.tyMotionStdTrav.tyBtnJogRear.bRtCompl	:= FALSE;
			tyP1031MagSetTeach.tyMotionStdTrav.tyBtnJogFront.bRtCompl	:= FALSE;
			tyP1031MagSetTeach.tyMotionStdTrav.tyBtnOrigin.bRtCompl		:= FALSE;
			tyP1031MagSetTeach.tyMotionStdTrav.tyBtnMovAbs.bRtCompl		:= FALSE;
			tyP1031MagSetTeach.tyMotionStdTrav.tyBtnMovRel.bRtCompl		:= FALSE;

			tyP1031MagSetTeach.tyTeachTravPosMag1.tyBtn2.bRtCompl		:= FALSE;
			tyP1031MagSetTeach.tyTeachTravPosMag2.tyBtn2.bRtCompl		:= FALSE;
			tyP1031MagSetTeach.tyTeachTravPosMag3.tyBtn2.bRtCompl		:= FALSE;
			tyP1031MagSetTeach.tyTeachTravPosMag4.tyBtn2.bRtCompl		:= FALSE;

			tyP1031MagSetTeach.tyMotionStdTrav.tyBtnStop.bValue			:= TRUE;
			tyP1031MagSetTeach.tyMotionStdTrav.tyBtnJogRear.bValue		:= FALSE;
			tyP1031MagSetTeach.tyMotionStdTrav.tyBtnJogFront.bValue		:= FALSE;
			tyP1031MagSetTeach.tyMotionStdTrav.tyBtnOrigin.bValue		:= FALSE;
			tyP1031MagSetTeach.tyMotionStdTrav.tyBtnMovAbs.bValue		:= FALSE;
			tyP1031MagSetTeach.tyMotionStdTrav.tyBtnMovRel.bValue		:= FALSE;

			tyP1031MagSetTeach.tyTeachTravPosMag1.tyBtn2.bValue			:= FALSE;
			tyP1031MagSetTeach.tyTeachTravPosMag2.tyBtn2.bValue			:= FALSE;
			tyP1031MagSetTeach.tyTeachTravPosMag3.tyBtn2.bValue			:= FALSE;
			tyP1031MagSetTeach.tyTeachTravPosMag4.tyBtn2.bValue			:= FALSE;

			tyP1031MagSetTeach.tyMotionStdTrav.tyBtnStop.bRtLk			:= TRUE;
			tyP1031MagSetTeach.tyMotionStdTrav.tyBtnJogRear.bRtLk		:= FALSE;
			tyP1031MagSetTeach.tyMotionStdTrav.tyBtnJogFront.bRtLk		:= FALSE;
			tyP1031MagSetTeach.tyMotionStdTrav.tyBtnOrigin.bRtLk		:= FALSE;
			tyP1031MagSetTeach.tyMotionStdTrav.tyBtnMovAbs.bRtLk		:= FALSE;
			tyP1031MagSetTeach.tyMotionStdTrav.tyBtnMovRel.bRtLk		:= FALSE;

			tyP1031MagSetTeach.tyTeachTravPosMag1.tyBtn2.bRtLk			:= FALSE;
			tyP1031MagSetTeach.tyTeachTravPosMag2.tyBtn2.bRtLk			:= FALSE;
			tyP1031MagSetTeach.tyTeachTravPosMag3.tyBtn2.bRtLk			:= FALSE;
			tyP1031MagSetTeach.tyTeachTravPosMag4.tyBtn2.bRtLk			:= FALSE;
		END_IF

	ELSIF (tyP1031MagSetTeach.tyMotionStdTrav.tyBtnJogRear.bRtCompl = TRUE) OR (tyP1031MagSetTeach.tyMotionStdTrav.tyBtnJogFront.bRtCompl = TRUE) OR (bJogStopTrav = TRUE) THEN
		bJogSlow					:= FALSE;
		bJogFast					:= FALSE;
		fbJogSlowToFastDlyTm.IN		:= FALSE;

		eTravAct		:= TravActJogStop;

		IF p_eTravStat = TravActJogStop AND p_eTravStatus = Done THEN
			eTravAct		:= TravActIdle;

			bJogStopTrav	:= FALSE;

			tyP1031MagSetTeach.tyMotionStdTrav.tyBtnStop.bRtCompl		:= FALSE;
			tyP1031MagSetTeach.tyMotionStdTrav.tyBtnJogRear.bRtCompl	:= FALSE;
			tyP1031MagSetTeach.tyMotionStdTrav.tyBtnJogFront.bRtCompl	:= FALSE;
			tyP1031MagSetTeach.tyMotionStdTrav.tyBtnOrigin.bRtCompl		:= FALSE;
			tyP1031MagSetTeach.tyMotionStdTrav.tyBtnMovAbs.bRtCompl		:= FALSE;
			tyP1031MagSetTeach.tyMotionStdTrav.tyBtnMovRel.bRtCompl		:= FALSE;

			tyP1031MagSetTeach.tyTeachTravPosMag1.tyBtn2.bRtCompl		:= FALSE;
			tyP1031MagSetTeach.tyTeachTravPosMag2.tyBtn2.bRtCompl		:= FALSE;
			tyP1031MagSetTeach.tyTeachTravPosMag3.tyBtn2.bRtCompl		:= FALSE;
			tyP1031MagSetTeach.tyTeachTravPosMag4.tyBtn2.bRtCompl		:= FALSE;

			tyP1031MagSetTeach.tyMotionStdTrav.tyBtnStop.bValue			:= TRUE;
			tyP1031MagSetTeach.tyMotionStdTrav.tyBtnJogRear.bValue		:= FALSE;
			tyP1031MagSetTeach.tyMotionStdTrav.tyBtnJogFront.bValue		:= FALSE;
			tyP1031MagSetTeach.tyMotionStdTrav.tyBtnOrigin.bValue		:= FALSE;
			tyP1031MagSetTeach.tyMotionStdTrav.tyBtnMovAbs.bValue		:= FALSE;
			tyP1031MagSetTeach.tyMotionStdTrav.tyBtnMovRel.bValue		:= FALSE;

			tyP1031MagSetTeach.tyTeachTravPosMag1.tyBtn2.bValue			:= FALSE;
			tyP1031MagSetTeach.tyTeachTravPosMag2.tyBtn2.bValue			:= FALSE;
			tyP1031MagSetTeach.tyTeachTravPosMag3.tyBtn2.bValue			:= FALSE;

			tyP1031MagSetTeach.tyMotionStdTrav.tyBtnStop.bRtLk			:= TRUE;
			tyP1031MagSetTeach.tyMotionStdTrav.tyBtnJogRear.bRtLk		:= FALSE;
			tyP1031MagSetTeach.tyMotionStdTrav.tyBtnJogFront.bRtLk		:= FALSE;
			tyP1031MagSetTeach.tyMotionStdTrav.tyBtnOrigin.bRtLk		:= FALSE;
			tyP1031MagSetTeach.tyMotionStdTrav.tyBtnMovAbs.bRtLk		:= FALSE;
			tyP1031MagSetTeach.tyMotionStdTrav.tyBtnMovRel.bRtLk		:= FALSE;

			tyP1031MagSetTeach.tyTeachTravPosMag1.tyBtn2.bRtLk			:= FALSE;
			tyP1031MagSetTeach.tyTeachTravPosMag2.tyBtn2.bRtLk			:= FALSE;
			tyP1031MagSetTeach.tyTeachTravPosMag3.tyBtn2.bRtLk			:= FALSE;
			tyP1031MagSetTeach.tyTeachTravPosMag4.tyBtn2.bRtLk			:= FALSE;

		END_IF

	ELSIF tyP1031MagSetTeach.tyMotionStdTrav.tyBtnPwr.bRtCompl = TRUE THEN
		tyP1031MagSetTeach.tyMotionStdTrav.tyBtnPwr.bRtLk				:= TRUE;

		IF tyP1031MagSetTeach.tyMotionStdTrav.tyBtnPwr.bValue = TRUE THEN
			eTravAct		:= TravActPwrOn;

			IF p_eTravStat = TravActPwrOn AND p_eTravStatus = Done THEN
				eTravAct	:= TravActIdle;

				tyP1031MagSetTeach.tyMotionStdTrav.tyBtnPwr.bRtCompl	:= FALSE;
				tyP1031MagSetTeach.tyMotionStdTrav.tyBtnPwr.bRtLk		:= FALSE;
			END_IF
		ELSE
			eTravAct		:= TravActPwrOff;

			IF p_eTravStat = TravActPwrOff AND p_eTravStatus = Done THEN
				eTravAct	:= TravActIdle;

				tyP1031MagSetTeach.tyMotionStdTrav.tyBtnPwr.bRtCompl		:= FALSE;
				tyP1031MagSetTeach.tyMotionStdTrav.tyBtnPwr.bRtLk		:= FALSE;
			END_IF
		END_IF

	ELSIF tyP1031MagSetTeach.tyMotionStdTrav.tyBtnOrigin.bRtCompl = TRUE THEN
		tyP1031MagSetTeach.tyMotionStdTrav.tyBtnOrigin.bValue			:= TRUE;
		tyP1031MagSetTeach.tyMotionStdTrav.tyBtnStop.bValue				:= FALSE;

		tyP1031MagSetTeach.tyMotionStdTrav.tyBtnOrigin.bRtLk				:= TRUE;
		tyP1031MagSetTeach.tyMotionStdTrav.tyBtnStop.bRtLk				:= FALSE;

		eTravAct		:= TravActHoming;

		IF p_eTravStat = TravActHoming AND p_eTravStatus = Done THEN
			eTravAct	:= TravActIdle;

			tyP1031MagSetTeach.tyMotionStdTrav.tyBtnOrigin.bRtCompl		:= FALSE;
			tyP1031MagSetTeach.tyMotionStdTrav.tyBtnOrigin.bValue		:= FALSE;
			tyP1031MagSetTeach.tyMotionStdTrav.tyBtnStop.bValue			:= TRUE;

			tyP1031MagSetTeach.tyMotionStdTrav.tyBtnOrigin.bRtLk		:= FALSE;
			tyP1031MagSetTeach.tyMotionStdTrav.tyBtnStop.bRtLk			:= TRUE;
		END_IF

	ELSIF tyP1031MagSetTeach.tyMotionStdTrav.tyBtnRst.bRtCompl = TRUE THEN
		tyP1031MagSetTeach.tyMotionStdTrav.tyBtnRst.bValue				:= TRUE;
		tyP1031MagSetTeach.tyMotionStdTrav.tyBtnRst.bRtLk				:= TRUE;

		eTravAct		:= TravActRstAxisErr;

		IF p_eTravStat = TravActRstAxisErr AND p_eTravStatus = Done THEN
			eTravAct	:= TravActIdle;

			tyP1031MagSetTeach.tyMotionStdTrav.tyBtnRst.bRtCompl		:= FALSE;
			tyP1031MagSetTeach.tyMotionStdTrav.tyBtnRst.bValue			:= FALSE;
			tyP1031MagSetTeach.tyMotionStdTrav.tyBtnRst.bRtLk			:= FALSE;

			fbLmtRstTm.IN			:= FALSE;
		END_IF

	ELSIF tyP1031MagSetTeach.tyTeachTravPosMag1.tyBtn2.bRtCompl = TRUE THEN
		tyP1031MagSetTeach.tyTeachTravPosMag1.tyBtn2.bValue		:= TRUE;
		tyP1031MagSetTeach.tyMotionStdTrav.tyBtnStop.bValue		:= FALSE;

		tyP1031MagSetTeach.tyTeachTravPosMag1.tyBtn2.bRtLk		:= TRUE;
		tyP1031MagSetTeach.tyMotionStdTrav.tyBtnStop.bRtLk		:= FALSE;

		diMnlTravNomSpd		:= tyP1031MagSetTeach.tyMotionStdTrav.tyNumNomSpd.diValue;

		eTravAct		:= TravActGoAPos;

		IF p_eTravStat = TravActGoAPos AND p_eTravStatus = Done THEN
			eTravAct	:= TravActIdle;

			tyP1031MagSetTeach.tyTeachTravPosMag1.tyBtn2.bRtCompl		:= FALSE;
			tyP1031MagSetTeach.tyTeachTravPosMag1.tyBtn2.bValue			:= FALSE;
			tyP1031MagSetTeach.tyMotionStdTrav.tyBtnStop.bValue			:= TRUE;

			tyP1031MagSetTeach.tyTeachTravPosMag1.tyBtn2.bRtLk			:= FALSE;
			tyP1031MagSetTeach.tyMotionStdTrav.tyBtnStop.bRtLk			:= TRUE;
		END_IF

	ELSIF tyP1031MagSetTeach.tyTeachTravPosMag2.tyBtn2.bRtCompl = TRUE THEN
		tyP1031MagSetTeach.tyTeachTravPosMag2.tyBtn2.bValue		:= TRUE;
		tyP1031MagSetTeach.tyMotionStdTrav.tyBtnStop.bValue		:= FALSE;

		tyP1031MagSetTeach.tyTeachTravPosMag2.tyBtn2.bRtLk		:= TRUE;
		tyP1031MagSetTeach.tyMotionStdTrav.tyBtnStop.bRtLk		:= FALSE;

		diMnlTravNomSpd		:= tyP1031MagSetTeach.tyMotionStdTrav.tyNumNomSpd.diValue;

		eTravAct		:= TravActGoBPos;

		IF p_eTravStat = TravActGoBPos AND p_eTravStatus = Done THEN
			eTravAct	:= TravActIdle;

			tyP1031MagSetTeach.tyTeachTravPosMag2.tyBtn2.bRtCompl		:= FALSE;
			tyP1031MagSetTeach.tyTeachTravPosMag2.tyBtn2.bValue			:= FALSE;
			tyP1031MagSetTeach.tyMotionStdTrav.tyBtnStop.bValue			:= TRUE;

			tyP1031MagSetTeach.tyTeachTravPosMag2.tyBtn2.bRtLk			:= FALSE;
			tyP1031MagSetTeach.tyMotionStdTrav.tyBtnStop.bRtLk			:= TRUE;
		END_IF

	ELSIF tyP1031MagSetTeach.tyTeachTravPosMag3.tyBtn2.bRtCompl = TRUE THEN
		tyP1031MagSetTeach.tyTeachTravPosMag3.tyBtn2.bValue		:= TRUE;
		tyP1031MagSetTeach.tyMotionStdTrav.tyBtnStop.bValue		:= FALSE;

		tyP1031MagSetTeach.tyTeachTravPosMag3.tyBtn2.bRtLk		:= TRUE;
		tyP1031MagSetTeach.tyMotionStdTrav.tyBtnStop.bRtLk		:= FALSE;

		diMnlTravNomSpd		:= tyP1031MagSetTeach.tyMotionStdTrav.tyNumNomSpd.diValue;

		eTravAct		:= TravActGoCPos;

		IF p_eTravStat = TravActGoCPos AND p_eTravStatus = Done THEN
			eTravAct	:= TravActIdle;

			tyP1031MagSetTeach.tyTeachTravPosMag3.tyBtn2.bRtCompl		:= FALSE;
			tyP1031MagSetTeach.tyTeachTravPosMag3.tyBtn2.bValue			:= FALSE;
			tyP1031MagSetTeach.tyMotionStdTrav.tyBtnStop.bValue			:= TRUE;

			tyP1031MagSetTeach.tyTeachTravPosMag3.tyBtn2.bRtLk			:= FALSE;
			tyP1031MagSetTeach.tyMotionStdTrav.tyBtnStop.bRtLk			:= TRUE;
		END_IF

	ELSIF tyP1031MagSetTeach.tyTeachTravPosMag4.tyBtn2.bRtCompl = TRUE THEN
		tyP1031MagSetTeach.tyTeachTravPosMag4.tyBtn2.bValue		:= TRUE;
		tyP1031MagSetTeach.tyMotionStdTrav.tyBtnStop.bValue		:= FALSE;

		tyP1031MagSetTeach.tyTeachTravPosMag4.tyBtn2.bRtLk		:= TRUE;
		tyP1031MagSetTeach.tyMotionStdTrav.tyBtnStop.bRtLk		:= FALSE;

		diMnlTravNomSpd		:= tyP1031MagSetTeach.tyMotionStdTrav.tyNumNomSpd.diValue;

		eTravAct		:= TravActGoGPos;

		IF p_eTravStat = TravActGoGPos AND p_eTravStatus = Done THEN
			eTravAct	:= TravActIdle;

			tyP1031MagSetTeach.tyTeachTravPosMag4.tyBtn2.bRtCompl		:= FALSE;
			tyP1031MagSetTeach.tyTeachTravPosMag4.tyBtn2.bValue			:= FALSE;
			tyP1031MagSetTeach.tyMotionStdTrav.tyBtnStop.bValue			:= TRUE;

			tyP1031MagSetTeach.tyTeachTravPosMag4.tyBtn2.bRtLk			:= FALSE;
			tyP1031MagSetTeach.tyMotionStdTrav.tyBtnStop.bRtLk			:= TRUE;
		END_IF

	ELSIF tyP1031MagSetTeach.tyMotionStdTrav.tyBtnMovAbs.bRtCompl = TRUE THEN
		tyP1031MagSetTeach.tyMotionStdTrav.tyBtnMovAbs.bValue			:= TRUE;
		tyP1031MagSetTeach.tyMotionStdTrav.tyBtnStop.bValue				:= FALSE;

		tyP1031MagSetTeach.tyMotionStdTrav.tyBtnMovAbs.bRtLk				:= TRUE;
		tyP1031MagSetTeach.tyMotionStdTrav.tyBtnStop.bRtLk				:= FALSE;

		diMnlTravTargetPos	:= tyP1031MagSetTeach.tyMotionStdTrav.tyNumTargetPos.diValue;
		diMnlTravNomSpd		:= tyP1031MagSetTeach.tyMotionStdTrav.tyNumNomSpd.diValue;

		eTravAct		:= TravActMovAbs;

		IF p_eTravStat = TravActMovAbs AND p_eTravStatus = Done THEN
			eTravAct	:= TravActIdle;

			tyP1031MagSetTeach.tyMotionStdTrav.tyBtnMovAbs.bRtCompl		:= FALSE;
			tyP1031MagSetTeach.tyMotionStdTrav.tyBtnMovAbs.bValue		:= FALSE;
			tyP1031MagSetTeach.tyMotionStdTrav.tyBtnStop.bValue			:= TRUE;

			tyP1031MagSetTeach.tyMotionStdTrav.tyBtnMovAbs.bRtLk			:= FALSE;
			tyP1031MagSetTeach.tyMotionStdTrav.tyBtnStop.bRtLk			:= TRUE;
		END_IF

	ELSIF tyP1031MagSetTeach.tyMotionStdTrav.tyBtnMovRel.bRtCompl = TRUE THEN
		tyP1031MagSetTeach.tyMotionStdTrav.tyBtnMovRel.bValue			:= TRUE;
		tyP1031MagSetTeach.tyMotionStdTrav.tyBtnStop.bValue				:= FALSE;

		tyP1031MagSetTeach.tyMotionStdTrav.tyBtnMovRel.bRtLk				:= TRUE;
		tyP1031MagSetTeach.tyMotionStdTrav.tyBtnStop.bRtLk				:= FALSE;

		diMnlTravStepSize	:= tyP1031MagSetTeach.tyMotionStdTrav.tyNumStepSize.diValue;
		diMnlTravNomSpd		:= tyP1031MagSetTeach.tyMotionStdTrav.tyNumNomSpd.diValue;

		eTravAct		:= TravActMovRel;

		IF p_eTravStat = TravActMovRel AND p_eTravStatus = Done THEN
			eTravAct	:= TravActIdle;

			tyP1031MagSetTeach.tyMotionStdTrav.tyBtnMovRel.bRtCompl		:= FALSE;
			tyP1031MagSetTeach.tyMotionStdTrav.tyBtnMovRel.bValue		:= FALSE;
			tyP1031MagSetTeach.tyMotionStdTrav.tyBtnStop.bValue			:= TRUE;

			tyP1031MagSetTeach.tyMotionStdTrav.tyBtnMovRel.bRtLk			:= FALSE;
			tyP1031MagSetTeach.tyMotionStdTrav.tyBtnStop.bRtLk			:= TRUE;
		END_IF

	ELSIF (tyP1031MagSetTeach.tyMotionStdTrav.tyBtnJogRear.bValue = TRUE) AND (fbJogSlowToFastDlyTm.Q = FALSE) AND (bJogSlow = FALSE) THEN
		tyP1031MagSetTeach.tyMotionStdTrav.tyBtnStop.bValue				:= FALSE;
		tyP1031MagSetTeach.tyMotionStdTrav.tyBtnStop.bRtLk				:= FALSE;

		fbJogSlowToFastDlyTm.IN		:= TRUE;

		diMnlTravJogSpd	:= tyP1031MagSetTeach.tyMotionStdTrav.tyNumSlwSpd.diValue;

		eTravAct		:= TravActJogRear;

		IF p_eTravStat = TravActJogRear AND p_eTravStatus = Done THEN
			eTravAct	:= TravActIdle;
			bJogSlow				:= TRUE;
		ELSIF p_eTravStatus = Error THEN
			fbJogSlowToFastDlyTm.IN	:= FALSE;
			bJogSlow				:= TRUE;
		END_IF

	ELSIF (tyP1031MagSetTeach.tyMotionStdTrav.tyBtnJogRear.bValue = TRUE) AND (fbJogSlowToFastDlyTm.Q = TRUE) AND (bJogFast = FALSE) THEN
		tyP1031MagSetTeach.tyMotionStdTrav.tyBtnStop.bValue					:= FALSE;
		tyP1031MagSetTeach.tyMotionStdTrav.tyBtnStop.bRtLk					:= FALSE;

		fbJogSlowToFastDlyTm.IN		:= TRUE;

		diMnlTravJogSpd	:= tyP1031MagSetTeach.tyMotionStdTrav.tyNumNomSpd.diValue;

		eTravAct		:= TravActJogRear;

		IF p_eTravStat = TravActJogRear AND p_eTravStatus = Done THEN
			eTravAct	:= TravActIdle;
			bJogFast				:= TRUE;
		ELSIF p_eTravStatus = Error THEN
			fbJogSlowToFastDlyTm.IN	:= FALSE;
			bJogFast				:= TRUE;
		END_IF

	ELSIF (tyP1031MagSetTeach.tyMotionStdTrav.tyBtnJogFront.bValue = TRUE) AND (fbJogSlowToFastDlyTm.Q = FALSE) AND (bJogSlow = FALSE) THEN
		tyP1031MagSetTeach.tyMotionStdTrav.tyBtnStop.bValue				:= FALSE;
		tyP1031MagSetTeach.tyMotionStdTrav.tyBtnStop.bRtLk				:= FALSE;

		fbJogSlowToFastDlyTm.IN		:= TRUE;

		diMnlTravJogSpd	:= tyP1031MagSetTeach.tyMotionStdTrav.tyNumSlwSpd.diValue;

		eTravAct		:= TravActJogFront;

		IF p_eTravStat = TravActJogFront AND p_eTravStatus = Done THEN
			eTravAct	:= TravActIdle;
			bJogSlow				:= TRUE;
		ELSIF p_eTravStatus = Error THEN
			fbJogSlowToFastDlyTm.IN	:= FALSE;
			bJogSlow				:= TRUE;
		END_IF

	ELSIF (tyP1031MagSetTeach.tyMotionStdTrav.tyBtnJogFront.bValue = TRUE) AND (fbJogSlowToFastDlyTm.Q = TRUE) AND (bJogFast = FALSE) THEN
		tyP1031MagSetTeach.tyMotionStdTrav.tyBtnStop.bValue				:= FALSE;
		tyP1031MagSetTeach.tyMotionStdTrav.tyBtnStop.bRtLk				:= FALSE;

		fbJogSlowToFastDlyTm.IN		:= TRUE;

		diMnlTravJogSpd	:= tyP1031MagSetTeach.tyMotionStdTrav.tyNumNomSpd.diValue;

		eTravAct		:= TravActJogFront;

		IF p_eTravStat = TravActJogFront AND p_eTravStatus = Done THEN
			eTravAct	:= TravActIdle;
			bJogFast	:= TRUE;
		ELSIF p_eTravStatus = Error THEN
			fbJogSlowToFastDlyTm.IN	:= FALSE;
			bJogFast				:= TRUE;
		END_IF
	END_IF

	IF tyP1031MagSetTeach.tyInOutletShutterFB.tyBtnOpen.bRtCompl = TRUE THEN
		tyP1031MagSetTeach.tyInOutletShutterFB.tyBtnOpen.bRtCompl	:= FALSE;

		tyP1031MagSetTeach.tyInOutletShutterFB.tyBtnOpen.bValue	:= TRUE;
		tyP1031MagSetTeach.tyInOutletShutterFB.tyBtnClose.bValue	:= FALSE;

	ELSIF tyP1031MagSetTeach.tyInOutletShutterFB.tyBtnClose.bRtCompl = TRUE THEN
		tyP1031MagSetTeach.tyInOutletShutterFB.tyBtnClose.bRtCompl	:= FALSE;

		tyP1031MagSetTeach.tyInOutletShutterFB.tyBtnClose.bValue	:= TRUE;
		tyP1031MagSetTeach.tyInOutletShutterFB.tyBtnOpen.bValue	:= FALSE;
	END_IF

	IF tyP1031MagSetTeach.tyInOutletShutterFB.tyBtnOpen.bValue = TRUE THEN
		eInShutterAct	:= PneuActRet;
		eInShutterAct2	:= PneuActRet;
		eInShutterAct3	:= PneuActRet;
		eOutShutterAct	:= PneuActRet;

		IF (p_eInShutterStat = PneuActRet AND p_eInShutterStatus = Done)
			AND (p_eInShutterStat2 = PneuActRet AND p_eInShutterStatus2 = Done)
			AND (p_eInShutterStat3 = PneuActRet AND p_eInShutterStatus3 = Done)
			AND (p_eOutShutterStat = PneuActRet AND p_eOutShutterStatus = Done)
			THEN
			eInShutterAct	:= PneuActIdle;
			eInShutterAct2	:= PneuActIdle;
			eInShutterAct3	:= PneuActIdle;
			eOutShutterAct	:= PneuActIdle;
			tyP1031MagSetTeach.tyInOutletShutterFB.tyBtnOpen.bValue	:= FALSE;
		ELSIF p_eInShutterStatus = Error OR p_eOutShutterStatus = Error THEN
			tyP1031MagSetTeach.tyInOutletShutterFB.tyBtnOpen.bValue	:= FALSE;
		END_IF

	ELSIF tyP1031MagSetTeach.tyInOutletShutterFB.tyBtnClose.bValue = TRUE THEN
		eInShutterAct	:= PneuActExt;
		eInShutterAct2	:= PneuActExt;
		eInShutterAct3	:= PneuActExt;
		eOutShutterAct	:= PneuActExt;
		IF (p_eInShutterStat = PneuActExt AND p_eInShutterStatus = Done)
			AND (p_eInShutterStat2 = PneuActExt AND p_eInShutterStatus2 = Done)
			AND (p_eInShutterStat3 = PneuActExt AND p_eInShutterStatus3 = Done)
			AND (p_eOutShutterStat = PneuActExt AND p_eOutShutterStatus = Done)
			THEN
			eInShutterAct	:= PneuActIdle;
			eInShutterAct2	:= PneuActIdle;
			eInShutterAct3	:= PneuActIdle;
			eOutShutterAct	:= PneuActIdle;
			tyP1031MagSetTeach.tyInOutletShutterFB.tyBtnClose.bValue := FALSE;
		ELSIF p_eInShutterStatus = Error OR p_eOutShutterStatus = Error THEN
			tyP1031MagSetTeach.tyInOutletShutterFB.tyBtnClose.bValue := FALSE;
		END_IF
	END_IF

	//bypass curtain sensor
	IF bTeachTravPosMag1 OR bTeachTravPosMag2 OR bTeachTravPosMag3 THEN
		bBypCurtainSen			:= tyP1031MagSetTeach.tyTeachTravPosMag1.tyBtn4.bValue OR tyP1031MagSetTeach.tyTeachTravPosMag2.tyBtn4.bValue OR tyP1031MagSetTeach.tyTeachTravPosMag3.tyBtn4.bValue;
		bBypCurtainPBLED		:= tyP1031MagSetTeach.tyTeachTravPosMag1.tyBtn4.bValue OR tyP1031MagSetTeach.tyTeachTravPosMag2.tyBtn4.bValue OR tyP1031MagSetTeach.tyTeachTravPosMag3.tyBtn4.bValue;
	END_IF

END_ACTION
```

#### Act_OptP1031TravMask.st
```iecst
ACTION Act_OptP1031TravMask:

	// Interlock Power
	IF p_bTravAxisErr = TRUE AND p_bTravPwrOn = FALSE THEN
		fUIInRtStatOff(ADR(tyP1031MagSetTeach.tyMotionStdTrav.tyBtnPwr.uiMaskRtStat));
		tyP1031MagSetTeach.tyMotionStdTrav.tyBtnPwr.bValue		:= FALSE;
	ELSE
		fUIInRtStatHide(ADR(tyP1031MagSetTeach.tyMotionStdTrav.tyBtnPwr.uiMaskRtStat));
	END_IF

	// Interlock Others Move
	IF p_bTravAxisErr = TRUE OR p_bTravPwrOn = FALSE THEN
		fUIInRtStatOff(ADR(tyP1031MagSetTeach.tyMotionStdTrav.tyBtnOrigin.uiMaskRtStat));
		fUIInRtStatOff(ADR(tyP1031MagSetTeach.tyMotionStdTrav.tyBtnMovRel.uiMaskRtStat));
		fUIInRtStatOff(ADR(tyP1031MagSetTeach.tyMotionStdTrav.tyBtnJogFront.uiMaskRtStat));
		fUIInRtStatOff(ADR(tyP1031MagSetTeach.tyMotionStdTrav.tyBtnJogRear.uiMaskRtStat));
	ELSE
		fUIInRtStatHide(ADR(tyP1031MagSetTeach.tyMotionStdTrav.tyBtnOrigin.uiMaskRtStat));
		fUIInRtStatHide(ADR(tyP1031MagSetTeach.tyMotionStdTrav.tyBtnMovRel.uiMaskRtStat));
		fUIInRtStatHide(ADR(tyP1031MagSetTeach.tyMotionStdTrav.tyBtnJogFront.uiMaskRtStat));
		fUIInRtStatHide(ADR(tyP1031MagSetTeach.tyMotionStdTrav.tyBtnJogRear.uiMaskRtStat));
	END_IF

	// Interlock Move Absolute
	IF p_bTravAxisErr = TRUE OR p_bTravPwrOn = FALSE OR p_bTravIsHomed = FALSE THEN
		fUIInRtStatOff(ADR(tyP1031MagSetTeach.tyTeachTravPosMag1.tyBtn2.uiMaskRtStat));
		fUIInRtStatOff(ADR(tyP1031MagSetTeach.tyTeachTravPosMag2.tyBtn2.uiMaskRtStat));
		fUIInRtStatOff(ADR(tyP1031MagSetTeach.tyTeachTravPosMag3.tyBtn2.uiMaskRtStat));
		fUIInRtStatOff(ADR(tyP1031MagSetTeach.tyTeachTravPosMag4.tyBtn2.uiMaskRtStat));
		fUIInRtStatOff(ADR(tyP1031MagSetTeach.tyMotionStdTrav.tyBtnMovAbs.uiMaskRtStat));
	ELSE
		fUIInRtStatHide(ADR(tyP1031MagSetTeach.tyTeachTravPosMag1.tyBtn2.uiMaskRtStat));
		fUIInRtStatHide(ADR(tyP1031MagSetTeach.tyTeachTravPosMag2.tyBtn2.uiMaskRtStat));
		fUIInRtStatHide(ADR(tyP1031MagSetTeach.tyTeachTravPosMag3.tyBtn2.uiMaskRtStat));
		fUIInRtStatHide(ADR(tyP1031MagSetTeach.tyTeachTravPosMag4.tyBtn2.uiMaskRtStat));
		fUIInRtStatHide(ADR(tyP1031MagSetTeach.tyMotionStdTrav.tyBtnMovAbs.uiMaskRtStat));
	END_IF

	//Interlock Limit Sensor
	IF tyP1031MagSetTeach.tyMotionStdTrav.tyBtnRearLmtSen.bValue = TRUE THEN
		fUIInRtStatOff(ADR(tyP1031MagSetTeach.tyMotionStdTrav.tyBtnJogRear.uiMaskRtStat));
	END_IF

	IF tyP1031MagSetTeach.tyMotionStdTrav.tyBtnFrontLmtSen.bValue = TRUE THEN
		fUIInRtStatOff(ADR(tyP1031MagSetTeach.tyMotionStdTrav.tyBtnJogFront.uiMaskRtStat));
	END_IF

	// Interlock When Moving
	IF tyP1031MagSetTeach.tyMotionStdTrav.tyBtnOrigin.bRtCompl = TRUE THEN
		fUIInRtStatOff(ADR(tyP1031MagSetTeach.tyMotionStdTrav.tyBtnMovAbs.uiMaskRtStat));
		fUIInRtStatOff(ADR(tyP1031MagSetTeach.tyMotionStdTrav.tyBtnMovRel.uiMaskRtStat));
		fUIInRtStatOff(ADR(tyP1031MagSetTeach.tyMotionStdTrav.tyBtnJogFront.uiMaskRtStat));
		fUIInRtStatOff(ADR(tyP1031MagSetTeach.tyMotionStdTrav.tyBtnJogRear.uiMaskRtStat));

		fUIInRtStatOff(ADR(tyP1031MagSetTeach.tyTeachTravPosMag1.tyBtn2.uiMaskRtStat));
		fUIInRtStatOff(ADR(tyP1031MagSetTeach.tyTeachTravPosMag2.tyBtn2.uiMaskRtStat));
		fUIInRtStatOff(ADR(tyP1031MagSetTeach.tyTeachTravPosMag3.tyBtn2.uiMaskRtStat));
		fUIInRtStatOff(ADR(tyP1031MagSetTeach.tyTeachTravPosMag4.tyBtn2.uiMaskRtStat));

	ELSIF tyP1031MagSetTeach.tyMotionStdTrav.tyBtnMovAbs.bRtCompl = TRUE THEN
		fUIInRtStatOff(ADR(tyP1031MagSetTeach.tyMotionStdTrav.tyBtnOrigin.uiMaskRtStat));
		fUIInRtStatOff(ADR(tyP1031MagSetTeach.tyMotionStdTrav.tyBtnMovRel.uiMaskRtStat));
		fUIInRtStatOff(ADR(tyP1031MagSetTeach.tyMotionStdTrav.tyBtnJogFront.uiMaskRtStat));
		fUIInRtStatOff(ADR(tyP1031MagSetTeach.tyMotionStdTrav.tyBtnJogRear.uiMaskRtStat));

		fUIInRtStatOff(ADR(tyP1031MagSetTeach.tyTeachTravPosMag1.tyBtn2.uiMaskRtStat));
		fUIInRtStatOff(ADR(tyP1031MagSetTeach.tyTeachTravPosMag2.tyBtn2.uiMaskRtStat));
		fUIInRtStatOff(ADR(tyP1031MagSetTeach.tyTeachTravPosMag3.tyBtn2.uiMaskRtStat));
		fUIInRtStatOff(ADR(tyP1031MagSetTeach.tyTeachTravPosMag4.tyBtn2.uiMaskRtStat));

	ELSIF tyP1031MagSetTeach.tyMotionStdTrav.tyBtnMovRel.bRtCompl = TRUE THEN
		fUIInRtStatOff(ADR(tyP1031MagSetTeach.tyMotionStdTrav.tyBtnOrigin.uiMaskRtStat));
		fUIInRtStatOff(ADR(tyP1031MagSetTeach.tyMotionStdTrav.tyBtnMovAbs.uiMaskRtStat));
		fUIInRtStatOff(ADR(tyP1031MagSetTeach.tyMotionStdTrav.tyBtnJogFront.uiMaskRtStat));
		fUIInRtStatOff(ADR(tyP1031MagSetTeach.tyMotionStdTrav.tyBtnJogRear.uiMaskRtStat));

		fUIInRtStatOff(ADR(tyP1031MagSetTeach.tyTeachTravPosMag1.tyBtn2.uiMaskRtStat));
		fUIInRtStatOff(ADR(tyP1031MagSetTeach.tyTeachTravPosMag2.tyBtn2.uiMaskRtStat));
		fUIInRtStatOff(ADR(tyP1031MagSetTeach.tyTeachTravPosMag3.tyBtn2.uiMaskRtStat));
		fUIInRtStatOff(ADR(tyP1031MagSetTeach.tyTeachTravPosMag4.tyBtn2.uiMaskRtStat));

	ELSIF tyP1031MagSetTeach.tyMotionStdTrav.tyBtnJogRear.bRtCompl = TRUE OR tyP1031MagSetTeach.tyMotionStdTrav.tyBtnJogRear.bValue = TRUE THEN
		fUIInRtStatOff(ADR(tyP1031MagSetTeach.tyMotionStdTrav.tyBtnOrigin.uiMaskRtStat));
		fUIInRtStatOff(ADR(tyP1031MagSetTeach.tyMotionStdTrav.tyBtnMovAbs.uiMaskRtStat));
		fUIInRtStatOff(ADR(tyP1031MagSetTeach.tyMotionStdTrav.tyBtnMovRel.uiMaskRtStat));
		fUIInRtStatOff(ADR(tyP1031MagSetTeach.tyMotionStdTrav.tyBtnJogFront.uiMaskRtStat));

		fUIInRtStatOff(ADR(tyP1031MagSetTeach.tyTeachTravPosMag1.tyBtn2.uiMaskRtStat));
		fUIInRtStatOff(ADR(tyP1031MagSetTeach.tyTeachTravPosMag2.tyBtn2.uiMaskRtStat));
		fUIInRtStatOff(ADR(tyP1031MagSetTeach.tyTeachTravPosMag3.tyBtn2.uiMaskRtStat));
		fUIInRtStatOff(ADR(tyP1031MagSetTeach.tyTeachTravPosMag4.tyBtn2.uiMaskRtStat));

	ELSIF tyP1031MagSetTeach.tyMotionStdTrav.tyBtnJogFront.bRtCompl = TRUE OR tyP1031MagSetTeach.tyMotionStdTrav.tyBtnJogFront.bValue = TRUE THEN
		fUIInRtStatOff(ADR(tyP1031MagSetTeach.tyMotionStdTrav.tyBtnOrigin.uiMaskRtStat));
		fUIInRtStatOff(ADR(tyP1031MagSetTeach.tyMotionStdTrav.tyBtnMovAbs.uiMaskRtStat));
		fUIInRtStatOff(ADR(tyP1031MagSetTeach.tyMotionStdTrav.tyBtnMovRel.uiMaskRtStat));
		fUIInRtStatOff(ADR(tyP1031MagSetTeach.tyMotionStdTrav.tyBtnJogRear.uiMaskRtStat));

		fUIInRtStatOff(ADR(tyP1031MagSetTeach.tyTeachTravPosMag1.tyBtn2.uiMaskRtStat));
		fUIInRtStatOff(ADR(tyP1031MagSetTeach.tyTeachTravPosMag2.tyBtn2.uiMaskRtStat));
		fUIInRtStatOff(ADR(tyP1031MagSetTeach.tyTeachTravPosMag3.tyBtn2.uiMaskRtStat));
		fUIInRtStatOff(ADR(tyP1031MagSetTeach.tyTeachTravPosMag4.tyBtn2.uiMaskRtStat));

	ELSIF tyP1031MagSetTeach.tyTeachTravPosMag1.tyBtn2.bRtCompl = TRUE THEN
		fUIInRtStatOff(ADR(tyP1031MagSetTeach.tyMotionStdTrav.tyBtnOrigin.uiMaskRtStat));
		fUIInRtStatOff(ADR(tyP1031MagSetTeach.tyMotionStdTrav.tyBtnMovAbs.uiMaskRtStat));
		fUIInRtStatOff(ADR(tyP1031MagSetTeach.tyMotionStdTrav.tyBtnMovRel.uiMaskRtStat));
		fUIInRtStatOff(ADR(tyP1031MagSetTeach.tyMotionStdTrav.tyBtnJogFront.uiMaskRtStat));
		fUIInRtStatOff(ADR(tyP1031MagSetTeach.tyMotionStdTrav.tyBtnJogRear.uiMaskRtStat));

	ELSIF tyP1031MagSetTeach.tyTeachTravPosMag2.tyBtn2.bRtCompl = TRUE THEN
		fUIInRtStatOff(ADR(tyP1031MagSetTeach.tyMotionStdTrav.tyBtnOrigin.uiMaskRtStat));
		fUIInRtStatOff(ADR(tyP1031MagSetTeach.tyMotionStdTrav.tyBtnMovAbs.uiMaskRtStat));
		fUIInRtStatOff(ADR(tyP1031MagSetTeach.tyMotionStdTrav.tyBtnMovRel.uiMaskRtStat));
		fUIInRtStatOff(ADR(tyP1031MagSetTeach.tyMotionStdTrav.tyBtnJogFront.uiMaskRtStat));
		fUIInRtStatOff(ADR(tyP1031MagSetTeach.tyMotionStdTrav.tyBtnJogRear.uiMaskRtStat));

	ELSIF tyP1031MagSetTeach.tyTeachTravPosMag3.tyBtn2.bRtCompl = TRUE THEN
		fUIInRtStatOff(ADR(tyP1031MagSetTeach.tyMotionStdTrav.tyBtnOrigin.uiMaskRtStat));
		fUIInRtStatOff(ADR(tyP1031MagSetTeach.tyMotionStdTrav.tyBtnMovAbs.uiMaskRtStat));
		fUIInRtStatOff(ADR(tyP1031MagSetTeach.tyMotionStdTrav.tyBtnMovRel.uiMaskRtStat));
		fUIInRtStatOff(ADR(tyP1031MagSetTeach.tyMotionStdTrav.tyBtnJogFront.uiMaskRtStat));
		fUIInRtStatOff(ADR(tyP1031MagSetTeach.tyMotionStdTrav.tyBtnJogRear.uiMaskRtStat));

	ELSIF tyP1031MagSetTeach.tyTeachTravPosMag4.tyBtn2.bRtCompl = TRUE THEN
		fUIInRtStatOff(ADR(tyP1031MagSetTeach.tyMotionStdTrav.tyBtnOrigin.uiMaskRtStat));
		fUIInRtStatOff(ADR(tyP1031MagSetTeach.tyMotionStdTrav.tyBtnMovAbs.uiMaskRtStat));
		fUIInRtStatOff(ADR(tyP1031MagSetTeach.tyMotionStdTrav.tyBtnMovRel.uiMaskRtStat));
		fUIInRtStatOff(ADR(tyP1031MagSetTeach.tyMotionStdTrav.tyBtnJogFront.uiMaskRtStat));
		fUIInRtStatOff(ADR(tyP1031MagSetTeach.tyMotionStdTrav.tyBtnJogRear.uiMaskRtStat));
	END_IF

	//Axis Error
	IF tyP1031MagSetTeach.tyMotionStdTrav.tyBtnPwr.bRtCompl = TRUE  THEN
		fUIInRtStatOff(ADR(tyP1031MagSetTeach.tyMotionStdTrav.tyBtnRst.uiMaskRtStat));
	ELSE
		fUIInRtStatHide(ADR(tyP1031MagSetTeach.tyMotionStdTrav.tyBtnRst.uiMaskRtStat));
	END_IF

	//Interlock Button Get
	IF p_bTravAxisErr = TRUE OR p_bTravIsHomed = FALSE OR p_bTravFwdLmtSen = TRUE OR p_bTravRevLmtSen = TRUE THEN
		fUIInRtStatOff(ADR(tyP1031MagSetTeach.tyTeachTravPosMag1.tyBtn1.uiMaskRtStat));
		fUIInRtStatOff(ADR(tyP1031MagSetTeach.tyTeachTravPosMag2.tyBtn1.uiMaskRtStat));
		fUIInRtStatOff(ADR(tyP1031MagSetTeach.tyTeachTravPosMag3.tyBtn1.uiMaskRtStat));
		fUIInRtStatOff(ADR(tyP1031MagSetTeach.tyTeachTravPosMag4.tyBtn1.uiMaskRtStat));
	ELSE
		fUIInRtStatHide(ADR(tyP1031MagSetTeach.tyTeachTravPosMag1.tyBtn1.uiMaskRtStat));
		fUIInRtStatHide(ADR(tyP1031MagSetTeach.tyTeachTravPosMag2.tyBtn1.uiMaskRtStat));
		fUIInRtStatHide(ADR(tyP1031MagSetTeach.tyTeachTravPosMag3.tyBtn1.uiMaskRtStat));
		fUIInRtStatHide(ADR(tyP1031MagSetTeach.tyTeachTravPosMag4.tyBtn1.uiMaskRtStat));
	END_IF

END_ACTION
```

#### Act_OptP1031TravUpdtDat.st
```iecst
ACTION Act_OptP1031TravUpdtDat:

	tyP1031MagSetTeach.tyMotionStdTrav.tyNumCurrPos.diValue			:= p_diTravActualPos;
	tyP1031MagSetTeach.tyMotionStdTrav.tyNumErrCode.diValue			:= UDINT_TO_DINT(p_udiTravAxisErrID);
	tyP1031MagSetTeach.tyMotionStdTrav.tyBitmapPwr.usiValueIdx		:= BOOL_TO_USINT(p_bTravPwrOn);
	tyP1031MagSetTeach.tyMotionStdTrav.tyBitmapRst.usiValueIdx		:= BOOL_TO_USINT(NOT p_bTravAxisErr);
	tyP1031MagSetTeach.tyMotionStdTrav.tyBitmapOrigin.usiValueIdx	:= BOOL_TO_USINT(p_bTravIsHomed);
	tyP1031MagSetTeach.tyMotionStdTrav.tyBtnFrontLmtSen.bValue		:= p_bTravFrontSen;
	tyP1031MagSetTeach.tyMotionStdTrav.tyBtnRearLmtSen.bValue		:= p_bTravRearSen;

	//Machine Bitmap
	IF   (p_tyNtParamCurr.eProjMag = LDMagDual AND p_tyNtParamCurr.bMagAutoVerifyPrep = FALSE)
		OR (p_tyNtParamCurr.eProjMag = LDMagTriple AND p_tyNtParamCurr.bMagAutoVerifyPrep = FALSE)
		OR (p_tyNtParamCurr.eProjMag = LDMagDual AND p_tyNtParamCurr.bMagAutoVerifyPrep = TRUE)
		THEN
		IF p_bTravIsHomed = TRUE THEN
			IF p_diTravActualPos <= (p_tyNtParamCurr.tyUITravTargetPos.diMax / 3) THEN
				tyP1031MagSetTeach.tyMotionStdTrav.tyBitmapMc.uiValueIdx 	:= 5;
			ELSIF p_diTravActualPos <= (p_tyNtParamCurr.tyUITravTargetPos.diMax / 3 * 2) THEN
				tyP1031MagSetTeach.tyMotionStdTrav.tyBitmapMc.uiValueIdx 	:= 6;
			ELSE
				tyP1031MagSetTeach.tyMotionStdTrav.tyBitmapMc.uiValueIdx 	:= 7;
			END_IF
		ELSE
			tyP1031MagSetTeach.tyMotionStdTrav.tyBitmapMc.uiValueIdx	:= 5;
		END_IF
	ELSIF p_tyNtParamCurr.eProjMag = LDMagTriple AND p_tyNtParamCurr.bMagAutoVerifyPrep = TRUE
		THEN
		IF p_bTravIsHomed = TRUE THEN
			IF p_diTravActualPos <= (p_tyNtParamCurr.tyUITravTargetPos.diMax / 3) THEN
				tyP1031MagSetTeach.tyMotionStdTrav.tyBitmapMc.uiValueIdx 	:= 26;
			ELSIF p_diTravActualPos <= (p_tyNtParamCurr.tyUITravTargetPos.diMax / 3 * 2) THEN
				tyP1031MagSetTeach.tyMotionStdTrav.tyBitmapMc.uiValueIdx 	:= 27;
			ELSE
				tyP1031MagSetTeach.tyMotionStdTrav.tyBitmapMc.uiValueIdx 	:= 28;
			END_IF
		ELSE
			tyP1031MagSetTeach.tyMotionStdTrav.tyBitmapMc.uiValueIdx	:= 26;
		END_IF
	ELSIF p_tyNtParamCurr.eProjMag = LDMagQuadruple AND p_tyNtParamCurr.bMagAutoVerifyPrep = TRUE
		THEN
		IF p_bTravIsHomed = TRUE THEN
			IF p_diTravActualPos <= (p_tyNtParamCurr.tyUITravTargetPos.diMax / 3) THEN
				tyP1031MagSetTeach.tyMotionStdTrav.tyBitmapMc.uiValueIdx 	:= 45;
			ELSIF p_diTravActualPos <= (p_tyNtParamCurr.tyUITravTargetPos.diMax / 3 * 2) THEN
				tyP1031MagSetTeach.tyMotionStdTrav.tyBitmapMc.uiValueIdx 	:= 46;
			ELSE
				tyP1031MagSetTeach.tyMotionStdTrav.tyBitmapMc.uiValueIdx 	:= 47;
			END_IF
		ELSE
			tyP1031MagSetTeach.tyMotionStdTrav.tyBitmapMc.uiValueIdx	:= 45;
		END_IF
	END_IF

	IF p_tyNtParamCurr.eProjMag = LDMagTriple AND p_tyNtParamCurr.bProjLifterMagPlatform THEN
		IF 	tyP1031MagSetTeach.tyMotionStdTrav.tyBitmapMc.uiValueIdx < 400 THEN
			tyP1031MagSetTeach.tyMotionStdTrav.tyBitmapMc.uiValueIdx	:= tyP1031MagSetTeach.tyMotionStdTrav.tyBitmapMc.uiValueIdx + 400;
		END_IF
	ELSIF p_tyNtParamCurr.eProjMag = LDMagTriple AND p_tyNtParamCurr.bMagAutoVerifyPrep = FALSE AND p_tyNtParamCurr.bProjMotorizedPullerPrep = FALSE THEN
		IF 	tyP1031MagSetTeach.tyMotionStdTrav.tyBitmapMc.uiValueIdx < 100 THEN
			tyP1031MagSetTeach.tyMotionStdTrav.tyBitmapMc.uiValueIdx	:= tyP1031MagSetTeach.tyMotionStdTrav.tyBitmapMc.uiValueIdx + 100;
		END_IF
	ELSIF p_tyNtParamCurr.eProjMag = LDMagDual AND p_tyNtParamCurr.bMagAutoVerifyPrep = FALSE THEN
		IF 	tyP1031MagSetTeach.tyMotionStdTrav.tyBitmapMc.uiValueIdx < 100 THEN
			IF p_tyNtParamCurr.sJobNo = '2023-0258A01' THEN
				tyP1031MagSetTeach.tyMotionStdTrav.tyBitmapMc.uiValueIdx	:= tyP1031MagSetTeach.tyMotionStdTrav.tyBitmapMc.uiValueIdx + 447-5;
			ELSE
				tyP1031MagSetTeach.tyMotionStdTrav.tyBitmapMc.uiValueIdx	:= tyP1031MagSetTeach.tyMotionStdTrav.tyBitmapMc.uiValueIdx + 200;
			END_IF
		END_IF
	ELSIF (p_tyNtParamCurr.eProjMag = LDMagDual OR p_tyNtParamCurr.eProjMag = LDMagTriple)
		AND p_tyNtParamCurr.bMagAutoVerifyPrep = TRUE THEN
		IF 	tyP1031MagSetTeach.tyMotionStdTrav.tyBitmapMc.uiValueIdx < 200 THEN
			tyP1031MagSetTeach.tyMotionStdTrav.tyBitmapMc.uiValueIdx	:= tyP1031MagSetTeach.tyMotionStdTrav.tyBitmapMc.uiValueIdx + 200;
		END_IF
	ELSIF p_tyNtParamCurr.eProjMag = LDMagTriple AND p_tyNtParamCurr.bMagAutoVerifyPrep = FALSE AND p_tyNtParamCurr.bProjMotorizedPullerPrep = TRUE THEN
		IF 	tyP1031MagSetTeach.tyMotionStdTrav.tyBitmapMc.uiValueIdx < 300 THEN
			tyP1031MagSetTeach.tyMotionStdTrav.tyBitmapMc.uiValueIdx	:= tyP1031MagSetTeach.tyMotionStdTrav.tyBitmapMc.uiValueIdx + 300;
		END_IF
	END_IF

END_ACTION
```

#### Act_OptP1031TravRstMnl.st
```iecst
ACTION Act_OptP1031TravRstMnl:

	IF EDGEPOS((bManualMod = FALSE) OR (p_eTravStatus = Error)) THEN

		bJogSlow				:= FALSE;
		bJogFast				:= FALSE;
		fbJogSlowToFastDlyTm.IN	:= FALSE;

		tyP1031MagSetTeach.tyMotionStdTrav.tyBtnPwr.bRtCompl			:= FALSE;
		tyP1031MagSetTeach.tyMotionStdTrav.tyBtnStop.bRtCompl			:= FALSE;
		tyP1031MagSetTeach.tyMotionStdTrav.tyBtnOrigin.bRtCompl			:= FALSE;
		tyP1031MagSetTeach.tyMotionStdTrav.tyBtnRst.bRtCompl			:= FALSE;
		tyP1031MagSetTeach.tyMotionStdTrav.tyBtnMovAbs.bRtCompl			:= FALSE;
		tyP1031MagSetTeach.tyMotionStdTrav.tyBtnMovRel.bRtCompl			:= FALSE;
		tyP1031MagSetTeach.tyMotionStdTrav.tyBtnJogFront.bRtCompl		:= FALSE;
		tyP1031MagSetTeach.tyMotionStdTrav.tyBtnJogRear.bRtCompl		:= FALSE;

		tyP1031MagSetTeach.tyTeachTravPosMag1.tyBtn2.bRtCompl			:= FALSE;
		tyP1031MagSetTeach.tyTeachTravPosMag2.tyBtn2.bRtCompl			:= FALSE;
		tyP1031MagSetTeach.tyTeachTravPosMag3.tyBtn2.bRtCompl			:= FALSE;
		tyP1031MagSetTeach.tyTeachTravPosMag4.tyBtn2.bRtCompl			:= FALSE;

		tyP1031MagSetTeach.tyMotionStdTrav.tyBtnPwr.bValue				:= FALSE;
		tyP1031MagSetTeach.tyMotionStdTrav.tyBtnStop.bValue				:= TRUE;
		tyP1031MagSetTeach.tyMotionStdTrav.tyBtnOrigin.bValue			:= FALSE;
		tyP1031MagSetTeach.tyMotionStdTrav.tyBtnRst.bValue				:= FALSE;
		tyP1031MagSetTeach.tyMotionStdTrav.tyBtnMovAbs.bValue			:= FALSE;
		tyP1031MagSetTeach.tyMotionStdTrav.tyBtnMovRel.bValue			:= FALSE;
		tyP1031MagSetTeach.tyMotionStdTrav.tyBtnJogFront.bValue			:= FALSE;
		tyP1031MagSetTeach.tyMotionStdTrav.tyBtnJogRear.bValue			:= FALSE;

		tyP1031MagSetTeach.tyTeachTravPosMag1.tyBtn2.bValue				:= FALSE;
		tyP1031MagSetTeach.tyTeachTravPosMag2.tyBtn2.bValue				:= FALSE;
		tyP1031MagSetTeach.tyTeachTravPosMag3.tyBtn2.bValue				:= FALSE;
		tyP1031MagSetTeach.tyTeachTravPosMag4.tyBtn2.bValue				:= FALSE;

		tyP1031MagSetTeach.tyMotionStdTrav.tyBtnPwr.bRtLk				:= FALSE;
		tyP1031MagSetTeach.tyMotionStdTrav.tyBtnStop.bRtLk				:= TRUE;
		tyP1031MagSetTeach.tyMotionStdTrav.tyBtnOrigin.bRtLk			:= FALSE;
		tyP1031MagSetTeach.tyMotionStdTrav.tyBtnRst.bRtLk				:= FALSE;
		tyP1031MagSetTeach.tyMotionStdTrav.tyBtnMovAbs.bRtLk			:= FALSE;
		tyP1031MagSetTeach.tyMotionStdTrav.tyBtnMovRel.bRtLk			:= FALSE;
		tyP1031MagSetTeach.tyMotionStdTrav.tyBtnJogFront.bRtLk			:= FALSE;
		tyP1031MagSetTeach.tyMotionStdTrav.tyBtnJogRear.bRtLk			:= FALSE;

		tyP1031MagSetTeach.tyTeachTravPosMag1.tyBtn2.bRtLk				:= FALSE;
		tyP1031MagSetTeach.tyTeachTravPosMag2.tyBtn2.bRtLk				:= FALSE;
		tyP1031MagSetTeach.tyTeachTravPosMag3.tyBtn2.bRtLk				:= FALSE;
		tyP1031MagSetTeach.tyTeachTravPosMag4.tyBtn2.bRtLk				:= FALSE;

		tyP1031MagSetTeach.tyMotionStdTrav.tyBtnPwr.uiMaskRtStat		:= TRUE;
		tyP1031MagSetTeach.tyMotionStdTrav.tyBtnOrigin.uiMaskRtStat		:= FALSE;
		tyP1031MagSetTeach.tyMotionStdTrav.tyBtnRst.uiMaskRtStat		:= TRUE;
		tyP1031MagSetTeach.tyMotionStdTrav.tyBtnMovAbs.uiMaskRtStat		:= FALSE;
		tyP1031MagSetTeach.tyMotionStdTrav.tyBtnMovRel.uiMaskRtStat		:= FALSE;
		tyP1031MagSetTeach.tyMotionStdTrav.tyBtnJogFront.uiMaskRtStat	:= FALSE;
		tyP1031MagSetTeach.tyMotionStdTrav.tyBtnJogRear.uiMaskRtStat	:= FALSE;

		tyP1031MagSetTeach.tyTeachTravPosMag1.tyBtn2.uiMaskRtStat		:= FALSE;
		tyP1031MagSetTeach.tyTeachTravPosMag2.tyBtn2.uiMaskRtStat		:= FALSE;
		tyP1031MagSetTeach.tyTeachTravPosMag3.tyBtn2.uiMaskRtStat		:= FALSE;
		tyP1031MagSetTeach.tyTeachTravPosMag4.tyBtn2.uiMaskRtStat		:= FALSE;

		eTravAct	:= TravActIdle;
	END_IF

END_ACTION
```

#### Act_OptP1031LifterTeach.st
```iecst
ACTION Act_OptP1031LifterTeach:

	IF tyP1031MagSetTeach.tyTeachLifterMag1Slt1Pos.tyBtn1.bRtCompl = TRUE THEN // Teach Lifter Magazine 1 Slot 1 Position

		p_tyC0008MsgBox ACCESS ADR(tyP1031MagSetTeach.tyMsgBoxUpdtLifterMag1Slt1Pos);

		IF tyP1031MagSetTeach.tyMsgBoxUpdtLifterMag1Slt1Pos.tyBtnNo.bRtCompl THEN
			tyP1031MagSetTeach.tyMsgBoxUpdtLifterMag1Slt1Pos.tyBtnNo.bRtCompl 	:= FALSE;
			tyP1031MagSetTeach.tyMsgBoxUpdtLifterMag1Slt1Pos.tyBtnNo.bValue 	:= FALSE;

			p_tyC0008MsgBox ACCESS ADR(tyP1031MagSetTeach.tyMsgBoxHide);

			//Write Actual Position To Magazine Setting.
			tyP1030MagSet.tyMagSet.tyNumLifterMag1Slt1Pos.diValue 	:= p_diLifterBtmActualPos;
			tyP1030MagSet.tyMagSet.tyNumLifterMag1Slt1Pos.bRtCompl	:= TRUE;

			//Back To Magazine Settings
			eChgPage	:= UIP1030MagSet;

			fUIInRtStatHide(ADR(tyP1030MagSet.tyMagSet.tyBtnSave.uiMaskRtStat));

			tyP1031MagSetTeach.tyTeachLifterMag1Slt1Pos.tyBtn1.bRtCompl	:= FALSE;
			tyP1031MagSetTeach.tyTeachLifterMag1Slt1Pos.tyBtn1.bValue	:= FALSE;

		END_IF

	ELSIF tyP1031MagSetTeach.tyTeachLifterMag2Slt1Pos.tyBtn1.bRtCompl = TRUE THEN // Teach Lifter Magazine 2 Slot 1 Position

		p_tyC0008MsgBox ACCESS ADR(tyP1031MagSetTeach.tyMsgBoxUpdtLifterMag2Slt1Pos);

		IF tyP1031MagSetTeach.tyMsgBoxUpdtLifterMag2Slt1Pos.tyBtnNo.bRtCompl THEN
			tyP1031MagSetTeach.tyMsgBoxUpdtLifterMag2Slt1Pos.tyBtnNo.bRtCompl 	:= FALSE;
			tyP1031MagSetTeach.tyMsgBoxUpdtLifterMag2Slt1Pos.tyBtnNo.bValue 	:= FALSE;

			p_tyC0008MsgBox ACCESS ADR(tyP1031MagSetTeach.tyMsgBoxHide);

			//Write Actual Position To Magazine Setting.
			tyP1030MagSet.tyMagSet.tyNumLifterMag2Slt1Pos.diValue 	:= p_diLifterBtmActualPos;
			tyP1030MagSet.tyMagSet.tyNumLifterMag2Slt1Pos.bRtCompl	:= TRUE;

			//Back To Magazine Settings
			eChgPage	:= UIP1030MagSet;

			fUIInRtStatHide(ADR(tyP1030MagSet.tyMagSet.tyBtnSave.uiMaskRtStat));

			tyP1031MagSetTeach.tyTeachLifterMag2Slt1Pos.tyBtn1.bRtCompl	:= FALSE;
			tyP1031MagSetTeach.tyTeachLifterMag2Slt1Pos.tyBtn1.bValue	:= FALSE;

		END_IF

	ELSIF tyP1031MagSetTeach.tyTeachLifterMag3Slt1Pos.tyBtn1.bRtCompl = TRUE THEN // Teach Lifter Magazine 3 Slot 1 Position

		p_tyC0008MsgBox ACCESS ADR(tyP1031MagSetTeach.tyMsgBoxUpdtLifterMag3Slt1Pos);

		IF tyP1031MagSetTeach.tyMsgBoxUpdtLifterMag3Slt1Pos.tyBtnNo.bRtCompl THEN
			tyP1031MagSetTeach.tyMsgBoxUpdtLifterMag3Slt1Pos.tyBtnNo.bRtCompl 	:= FALSE;
			tyP1031MagSetTeach.tyMsgBoxUpdtLifterMag3Slt1Pos.tyBtnNo.bValue 	:= FALSE;

			p_tyC0008MsgBox ACCESS ADR(tyP1031MagSetTeach.tyMsgBoxHide);

			//Write Actual Position To Magazine Setting.
			tyP1030MagSet.tyMagSet.tyNumLifterMag3Slt1Pos.diValue 	:= p_diLifterBtmActualPos;
			tyP1030MagSet.tyMagSet.tyNumLifterMag3Slt1Pos.bRtCompl	:= TRUE;

			//Back To Magazine Settings
			eChgPage	:= UIP1030MagSet;

			fUIInRtStatHide(ADR(tyP1030MagSet.tyMagSet.tyBtnSave.uiMaskRtStat));

			tyP1031MagSetTeach.tyTeachLifterMag3Slt1Pos.tyBtn1.bRtCompl	:= FALSE;
			tyP1031MagSetTeach.tyTeachLifterMag3Slt1Pos.tyBtn1.bValue	:= FALSE;

		END_IF

	ELSIF tyP1031MagSetTeach.tyTeachLifterMag4Slt1Pos.tyBtn1.bRtCompl = TRUE THEN // Teach Lifter Magazine 4 Slot 1 Position

		p_tyC0008MsgBox ACCESS ADR(tyP1031MagSetTeach.tyMsgBoxUpdtLifterMag4Slt1Pos);

		IF tyP1031MagSetTeach.tyMsgBoxUpdtLifterMag4Slt1Pos.tyBtnNo.bRtCompl THEN
			tyP1031MagSetTeach.tyMsgBoxUpdtLifterMag4Slt1Pos.tyBtnNo.bRtCompl 	:= FALSE;
			tyP1031MagSetTeach.tyMsgBoxUpdtLifterMag4Slt1Pos.tyBtnNo.bValue 	:= FALSE;

			p_tyC0008MsgBox ACCESS ADR(tyP1031MagSetTeach.tyMsgBoxHide);

			//Write Actual Position To Magazine Setting.
			tyP1030MagSet.tyMagSet.tyNumLifterMag4Slt1Pos.diValue 	:= p_diLifterBtmActualPos;
			tyP1030MagSet.tyMagSet.tyNumLifterMag4Slt1Pos.bRtCompl	:= TRUE;

			//Back To Magazine Settings
			eChgPage	:= UIP1030MagSet;

			fUIInRtStatHide(ADR(tyP1030MagSet.tyMagSet.tyBtnSave.uiMaskRtStat));

			tyP1031MagSetTeach.tyTeachLifterMag4Slt1Pos.tyBtn1.bRtCompl	:= FALSE;
			tyP1031MagSetTeach.tyTeachLifterMag4Slt1Pos.tyBtn1.bValue	:= FALSE;

		END_IF
	END_IF

END_ACTION
```

#### Act_OptP1031LifterFBCtrl.st
```iecst
ACTION Act_OptP1031LifterFBCtrl:

	fbJogSlowToFastDlyTm.PT	:= T#2s;
	fbJogSlowToFastDlyTm;
	fbLmtRstTm;

	//Lifter Safety Sensor Interruption
	IF EDGENEG(p_tyDI.bLifterSafetyLmtSW1 AND p_tyDI.bLifterSafetyLmtSW2 AND p_tyDI.bLifterTimingBeltSen) THEN
		tyP1031MagSetTeach.tyMotionStdLifter.tyBtnStop.bRtCompl	:= TRUE;
	END_IF

//	IF EDGEPOS((p_udiLifterBtmAxisErrID = 21570 OR p_udiLifterBtmAxisErrID = 21571) AND tyP1031MagSetTeach.tyMotionStdLifter.tyBtnJogDown.bValue = FALSE AND tyP1031MagSetTeach.tyMotionStdLifter.tyBtnJogUp.bValue = FALSE) THEN
	IF EDGEPOS((p_bLifterBtmFwdLmtSen OR p_bLifterBtmRevLmtSen OR p_udiLifterBtmAxisErrID = 21570 OR p_udiLifterBtmAxisErrID = 21571)
		AND tyP1026McSetTeach.tyMotionStdLifter.tyBtnJogDown.bValue = FALSE
		AND tyP1026McSetTeach.tyMotionStdLifter.tyBtnJogUp.bValue = FALSE) THEN
			fbLmtRstTm.IN				:= TRUE;
	END_IF

	IF fbLmtRstTm.Q = TRUE THEN
		tyP1031MagSetTeach.tyMotionStdLifter.tyBtnRst.bRtCompl		:= TRUE;
	END_IF

	IF (tyP1031MagSetTeach.tyMotionStdLifter.tyBtnJogUp.bValue = FALSE AND tyP1031MagSetTeach.tyMotionStdLifter.tyBtnJogDown.bValue = FALSE) AND (p_bLifterBtmJogging = TRUE) THEN
		bJogStopLifter	:= TRUE;
	END_IF

	IF tyP1031MagSetTeach.tyMotionStdLifter.tyBtnStop.bRtCompl = TRUE THEN
		eLifterBtmAct		:= LifterActStop;

		IF p_eLifterBtmStat = LifterActStop AND p_eLifterBtmStatus = Done THEN
			eLifterBtmAct	:= LifterActIdle;

			tyP1031MagSetTeach.tyMotionStdLifter.tyBtnStop.bRtCompl			:= FALSE;
			tyP1031MagSetTeach.tyMotionStdLifter.tyBtnJogDown.bRtCompl		:= FALSE;
			tyP1031MagSetTeach.tyMotionStdLifter.tyBtnJogUp.bRtCompl		:= FALSE;
			tyP1031MagSetTeach.tyMotionStdLifter.tyBtnOrigin.bRtCompl		:= FALSE;
			tyP1031MagSetTeach.tyMotionStdLifter.tyBtnMovAbs.bRtCompl		:= FALSE;
			tyP1031MagSetTeach.tyMotionStdLifter.tyBtnMovRel.bRtCompl		:= FALSE;

			tyP1031MagSetTeach.tyTeachLifterMag1Slt1Pos.tyBtn2.bRtCompl		:= FALSE;
			tyP1031MagSetTeach.tyTeachLifterMag2Slt1Pos.tyBtn2.bRtCompl		:= FALSE;
			tyP1031MagSetTeach.tyTeachLifterMag3Slt1Pos.tyBtn2.bRtCompl		:= FALSE;
			tyP1031MagSetTeach.tyTeachLifterMag4Slt1Pos.tyBtn2.bRtCompl		:= FALSE;

			tyP1031MagSetTeach.tyMotionStdLifter.tyBtnStop.bValue			:= TRUE;
			tyP1031MagSetTeach.tyMotionStdLifter.tyBtnJogDown.bValue		:= FALSE;
			tyP1031MagSetTeach.tyMotionStdLifter.tyBtnJogUp.bValue			:= FALSE;
			tyP1031MagSetTeach.tyMotionStdLifter.tyBtnOrigin.bValue			:= FALSE;
			tyP1031MagSetTeach.tyMotionStdLifter.tyBtnMovAbs.bValue			:= FALSE;
			tyP1031MagSetTeach.tyMotionStdLifter.tyBtnMovRel.bValue			:= FALSE;

			tyP1031MagSetTeach.tyTeachLifterMag1Slt1Pos.tyBtn2.bValue		:= FALSE;
			tyP1031MagSetTeach.tyTeachLifterMag2Slt1Pos.tyBtn2.bValue		:= FALSE;
			tyP1031MagSetTeach.tyTeachLifterMag3Slt1Pos.tyBtn2.bValue		:= FALSE;
			tyP1031MagSetTeach.tyTeachLifterMag4Slt1Pos.tyBtn2.bValue		:= FALSE;

			tyP1031MagSetTeach.tyMotionStdLifter.tyBtnStop.bRtLk			:= TRUE;
			tyP1031MagSetTeach.tyMotionStdLifter.tyBtnJogDown.bRtLk			:= FALSE;
			tyP1031MagSetTeach.tyMotionStdLifter.tyBtnJogUp.bRtLk			:= FALSE;
			tyP1031MagSetTeach.tyMotionStdLifter.tyBtnOrigin.bRtLk			:= FALSE;
			tyP1031MagSetTeach.tyMotionStdLifter.tyBtnMovAbs.bRtLk			:= FALSE;
			tyP1031MagSetTeach.tyMotionStdLifter.tyBtnMovRel.bRtLk			:= FALSE;

			tyP1031MagSetTeach.tyTeachLifterMag1Slt1Pos.tyBtn2.bRtLk		:= FALSE;
			tyP1031MagSetTeach.tyTeachLifterMag2Slt1Pos.tyBtn2.bRtLk		:= FALSE;
			tyP1031MagSetTeach.tyTeachLifterMag3Slt1Pos.tyBtn2.bRtLk		:= FALSE;
			tyP1031MagSetTeach.tyTeachLifterMag4Slt1Pos.tyBtn2.bRtLk		:= FALSE;
		END_IF

	ELSIF (tyP1031MagSetTeach.tyMotionStdLifter.tyBtnJogDown.bRtCompl = TRUE) OR (tyP1031MagSetTeach.tyMotionStdLifter.tyBtnJogUp.bRtCompl = TRUE) OR (bJogStopLifter = TRUE) THEN
		bJogSlow					:= FALSE;
		bJogFast					:= FALSE;
		fbJogSlowToFastDlyTm.IN		:= FALSE;

		eLifterBtmAct		:= LifterActJogStop;

		IF p_eLifterBtmStat = LifterActJogStop AND p_eLifterBtmStatus = Done THEN
			eLifterBtmAct		:= LifterActIdle;

			bJogStopLifter	:= FALSE;

			tyP1031MagSetTeach.tyMotionStdLifter.tyBtnStop.bRtCompl			:= FALSE;
			tyP1031MagSetTeach.tyMotionStdLifter.tyBtnJogDown.bRtCompl		:= FALSE;
			tyP1031MagSetTeach.tyMotionStdLifter.tyBtnJogUp.bRtCompl		:= FALSE;
			tyP1031MagSetTeach.tyMotionStdLifter.tyBtnOrigin.bRtCompl		:= FALSE;
			tyP1031MagSetTeach.tyMotionStdLifter.tyBtnMovAbs.bRtCompl		:= FALSE;
			tyP1031MagSetTeach.tyMotionStdLifter.tyBtnMovRel.bRtCompl		:= FALSE;

			tyP1031MagSetTeach.tyTeachLifterMag1Slt1Pos.tyBtn2.bRtCompl		:= FALSE;
			tyP1031MagSetTeach.tyTeachLifterMag2Slt1Pos.tyBtn2.bRtCompl		:= FALSE;
			tyP1031MagSetTeach.tyTeachLifterMag3Slt1Pos.tyBtn2.bRtCompl		:= FALSE;
			tyP1031MagSetTeach.tyTeachLifterMag4Slt1Pos.tyBtn2.bRtCompl		:= FALSE;

			tyP1031MagSetTeach.tyMotionStdLifter.tyBtnStop.bValue			:= TRUE;
			tyP1031MagSetTeach.tyMotionStdLifter.tyBtnJogDown.bValue		:= FALSE;
			tyP1031MagSetTeach.tyMotionStdLifter.tyBtnJogUp.bValue			:= FALSE;
			tyP1031MagSetTeach.tyMotionStdLifter.tyBtnOrigin.bValue			:= FALSE;
			tyP1031MagSetTeach.tyMotionStdLifter.tyBtnMovAbs.bValue			:= FALSE;
			tyP1031MagSetTeach.tyMotionStdLifter.tyBtnMovRel.bValue			:= FALSE;

			tyP1031MagSetTeach.tyTeachLifterMag1Slt1Pos.tyBtn2.bValue		:= FALSE;
			tyP1031MagSetTeach.tyTeachLifterMag2Slt1Pos.tyBtn2.bValue		:= FALSE;
			tyP1031MagSetTeach.tyTeachLifterMag3Slt1Pos.tyBtn2.bValue		:= FALSE;
			tyP1031MagSetTeach.tyTeachLifterMag4Slt1Pos.tyBtn2.bValue		:= FALSE;

			tyP1031MagSetTeach.tyMotionStdLifter.tyBtnStop.bRtLk			:= TRUE;
			tyP1031MagSetTeach.tyMotionStdLifter.tyBtnJogDown.bRtLk			:= FALSE;
			tyP1031MagSetTeach.tyMotionStdLifter.tyBtnJogUp.bRtLk			:= FALSE;
			tyP1031MagSetTeach.tyMotionStdLifter.tyBtnOrigin.bRtLk			:= FALSE;
			tyP1031MagSetTeach.tyMotionStdLifter.tyBtnMovAbs.bRtLk			:= FALSE;
			tyP1031MagSetTeach.tyMotionStdLifter.tyBtnMovRel.bRtLk			:= FALSE;

			tyP1031MagSetTeach.tyTeachLifterMag1Slt1Pos.tyBtn2.bRtLk		:= FALSE;
			tyP1031MagSetTeach.tyTeachLifterMag2Slt1Pos.tyBtn2.bRtLk		:= FALSE;
			tyP1031MagSetTeach.tyTeachLifterMag3Slt1Pos.tyBtn2.bRtLk		:= FALSE;
			tyP1031MagSetTeach.tyTeachLifterMag4Slt1Pos.tyBtn2.bRtLk		:= FALSE;
		END_IF

	ELSIF tyP1031MagSetTeach.tyMotionStdLifter.tyBtnPwr.bRtCompl = TRUE THEN
		tyP1031MagSetTeach.tyMotionStdLifter.tyBtnPwr.bRtLk					:= TRUE;

		IF tyP1031MagSetTeach.tyMotionStdLifter.tyBtnPwr.bValue = TRUE THEN
			eLifterBtmAct		:= LifterActPwrOn;

			IF p_eLifterBtmStat = LifterActPwrOn AND p_eLifterBtmStatus = Done THEN
				eLifterBtmAct	:= LifterActIdle;

				tyP1031MagSetTeach.tyMotionStdLifter.tyBtnPwr.bRtCompl		:= FALSE;
				tyP1031MagSetTeach.tyMotionStdLifter.tyBtnPwr.bRtLk		:= FALSE;
			END_IF
		ELSE
			eLifterBtmAct		:= LifterActPwrOff;

			IF p_eLifterBtmStat = LifterActPwrOff AND p_eLifterBtmStatus = Done THEN
				eLifterBtmAct	:= LifterActIdle;

				tyP1031MagSetTeach.tyMotionStdLifter.tyBtnPwr.bRtCompl		:= FALSE;
				tyP1031MagSetTeach.tyMotionStdLifter.tyBtnPwr.bRtLk		:= FALSE;
			END_IF
		END_IF

	ELSIF tyP1031MagSetTeach.tyMotionStdLifter.tyBtnOrigin.bRtCompl = TRUE THEN
		tyP1031MagSetTeach.tyMotionStdLifter.tyBtnOrigin.bValue				:= TRUE;
		tyP1031MagSetTeach.tyMotionStdLifter.tyBtnStop.bValue					:= FALSE;

		tyP1031MagSetTeach.tyMotionStdLifter.tyBtnOrigin.bRtLk					:= TRUE;
		tyP1031MagSetTeach.tyMotionStdLifter.tyBtnStop.bRtLk					:= FALSE;

		eLifterBtmAct		:= LifterActHoming;

		IF p_eLifterBtmStat = LifterActHoming AND p_eLifterBtmStatus = Done THEN
			eLifterBtmAct	:= LifterActIdle;

			tyP1031MagSetTeach.tyMotionStdLifter.tyBtnOrigin.bRtCompl		:= FALSE;
			tyP1031MagSetTeach.tyMotionStdLifter.tyBtnOrigin.bValue		:= FALSE;
			tyP1031MagSetTeach.tyMotionStdLifter.tyBtnStop.bValue			:= TRUE;

			tyP1031MagSetTeach.tyMotionStdLifter.tyBtnOrigin.bRtLk			:= FALSE;
			tyP1031MagSetTeach.tyMotionStdLifter.tyBtnStop.bRtLk			:= TRUE;

		END_IF

	ELSIF tyP1031MagSetTeach.tyMotionStdLifter.tyBtnRst.bRtCompl = TRUE THEN
		tyP1031MagSetTeach.tyMotionStdLifter.tyBtnRst.bValue				:= TRUE;
		tyP1031MagSetTeach.tyMotionStdLifter.tyBtnRst.bRtLk				:= TRUE;

		eLifterBtmAct		:= LifterActRstAxisErr;

		IF p_eLifterBtmStat = LifterActRstAxisErr AND p_eLifterBtmStatus = Done THEN
			eLifterBtmAct	:= LifterActIdle;

			tyP1031MagSetTeach.tyMotionStdLifter.tyBtnRst.bRtCompl			:= FALSE;
			tyP1031MagSetTeach.tyMotionStdLifter.tyBtnRst.bValue			:= FALSE;
			tyP1031MagSetTeach.tyMotionStdLifter.tyBtnRst.bRtLk			:= FALSE;

			fbLmtRstTm.IN			:= FALSE;
		END_IF

	ELSIF tyP1031MagSetTeach.tyTeachLifterMag1Slt1Pos.tyBtn2.bRtCompl = TRUE THEN
		tyP1031MagSetTeach.tyTeachLifterMag1Slt1Pos.tyBtn2.bValue			:= TRUE;
		tyP1031MagSetTeach.tyMotionStdLifter.tyBtnStop.bValue				:= FALSE;

		tyP1031MagSetTeach.tyTeachLifterMag1Slt1Pos.tyBtn2.bRtLk		:= TRUE;
		tyP1031MagSetTeach.tyMotionStdLifter.tyBtnStop.bRtLk			:= FALSE;

		//diMnlLifterMag1GoSlt	:= 1;
		diMnlLifterMag1GoSlt	:= tyP1031MagSetTeach.tyTeachLifterMag1Slt1Pos.tyNumNewSlt.diValue;
		diMnlLifterNomSpd		:= tyP1031MagSetTeach.tyMotionStdLifter.tyNumNomSpd.diValue;

		eLifterBtmAct		:= LifterActGoASltPos;

		IF p_eLifterBtmStat = LifterActGoASltPos AND p_eLifterBtmStatus = Done THEN
			eLifterBtmAct	:= LifterActIdle;

			tyP1031MagSetTeach.tyTeachLifterMag1Slt1Pos.tyBtn2.bRtCompl			:= FALSE;
			tyP1031MagSetTeach.tyTeachLifterMag1Slt1Pos.tyBtn2.bValue			:= FALSE;
			tyP1031MagSetTeach.tyMotionStdLifter.tyBtnStop.bValue				:= TRUE;

			tyP1031MagSetTeach.tyTeachLifterMag1Slt1Pos.tyBtn2.bRtLk			:= FALSE;
			tyP1031MagSetTeach.tyMotionStdLifter.tyBtnStop.bRtLk				:= TRUE;
		END_IF

	ELSIF tyP1031MagSetTeach.tyTeachLifterMag2Slt1Pos.tyBtn2.bRtCompl = TRUE THEN
		tyP1031MagSetTeach.tyTeachLifterMag2Slt1Pos.tyBtn2.bValue			:= TRUE;
		tyP1031MagSetTeach.tyMotionStdLifter.tyBtnStop.bValue				:= FALSE;

		tyP1031MagSetTeach.tyTeachLifterMag2Slt1Pos.tyBtn2.bRtLk			:= TRUE;
		tyP1031MagSetTeach.tyMotionStdLifter.tyBtnStop.bRtLk				:= FALSE;

		//diMnlLifterMag2GoSlt	:= 1;
		diMnlLifterMag2GoSlt	:= tyP1031MagSetTeach.tyTeachLifterMag2Slt1Pos.tyNumNewSlt.diValue;
		diMnlLifterNomSpd		:= tyP1031MagSetTeach.tyMotionStdLifter.tyNumNomSpd.diValue;

		eLifterBtmAct		:= LifterActGoBSltPos;

		IF p_eLifterBtmStat = LifterActGoBSltPos AND p_eLifterBtmStatus = Done THEN
			eLifterBtmAct	:= LifterActIdle;

			tyP1031MagSetTeach.tyTeachLifterMag2Slt1Pos.tyBtn2.bRtCompl			:= FALSE;
			tyP1031MagSetTeach.tyTeachLifterMag2Slt1Pos.tyBtn2.bValue			:= FALSE;
			tyP1031MagSetTeach.tyMotionStdLifter.tyBtnStop.bValue				:= TRUE;

			tyP1031MagSetTeach.tyTeachLifterMag2Slt1Pos.tyBtn2.bRtLk			:= FALSE;
			tyP1031MagSetTeach.tyMotionStdLifter.tyBtnStop.bRtLk				:= TRUE;
		END_IF

	ELSIF tyP1031MagSetTeach.tyTeachLifterMag3Slt1Pos.tyBtn2.bRtCompl = TRUE THEN
		tyP1031MagSetTeach.tyTeachLifterMag3Slt1Pos.tyBtn2.bValue			:= TRUE;
		tyP1031MagSetTeach.tyMotionStdLifter.tyBtnStop.bValue				:= FALSE;

		tyP1031MagSetTeach.tyTeachLifterMag3Slt1Pos.tyBtn2.bRtLk			:= TRUE;
		tyP1031MagSetTeach.tyMotionStdLifter.tyBtnStop.bRtLk				:= FALSE;

		//diMnlLifterMag3GoSlt	:= 1;
		diMnlLifterMag3GoSlt	:= tyP1031MagSetTeach.tyTeachLifterMag3Slt1Pos.tyNumNewSlt.diValue;
		diMnlLifterNomSpd		:= tyP1031MagSetTeach.tyMotionStdLifter.tyNumNomSpd.diValue;

		eLifterBtmAct		:= LifterActGoCSltPos;

		IF p_eLifterBtmStat = LifterActGoCSltPos AND p_eLifterBtmStatus = Done THEN
			eLifterBtmAct	:= LifterActIdle;

			tyP1031MagSetTeach.tyTeachLifterMag3Slt1Pos.tyBtn2.bRtCompl			:= FALSE;
			tyP1031MagSetTeach.tyTeachLifterMag3Slt1Pos.tyBtn2.bValue			:= FALSE;
			tyP1031MagSetTeach.tyMotionStdLifter.tyBtnStop.bValue				:= TRUE;

			tyP1031MagSetTeach.tyTeachLifterMag3Slt1Pos.tyBtn2.bRtLk			:= FALSE;
			tyP1031MagSetTeach.tyMotionStdLifter.tyBtnStop.bRtLk				:= TRUE;
		END_IF

	ELSIF tyP1031MagSetTeach.tyTeachLifterMag4Slt1Pos.tyBtn2.bRtCompl = TRUE THEN
		tyP1031MagSetTeach.tyTeachLifterMag4Slt1Pos.tyBtn2.bValue			:= TRUE;
		tyP1031MagSetTeach.tyMotionStdLifter.tyBtnStop.bValue				:= FALSE;

		tyP1031MagSetTeach.tyTeachLifterMag4Slt1Pos.tyBtn2.bRtLk			:= TRUE;
		tyP1031MagSetTeach.tyMotionStdLifter.tyBtnStop.bRtLk				:= FALSE;

		//diMnlLifterMag4GoSlt	:= 1;
		diMnlLifterMag4GoSlt	:= tyP1031MagSetTeach.tyTeachLifterMag4Slt1Pos.tyNumNewSlt.diValue;
		diMnlLifterNomSpd		:= tyP1031MagSetTeach.tyMotionStdLifter.tyNumNomSpd.diValue;

		eLifterBtmAct		:= LifterActGoDSltPos;

		IF p_eLifterBtmStat = LifterActGoDSltPos AND p_eLifterBtmStatus = Done THEN
			eLifterBtmAct	:= LifterActIdle;

			tyP1031MagSetTeach.tyTeachLifterMag4Slt1Pos.tyBtn2.bRtCompl			:= FALSE;
			tyP1031MagSetTeach.tyTeachLifterMag4Slt1Pos.tyBtn2.bValue			:= FALSE;
			tyP1031MagSetTeach.tyMotionStdLifter.tyBtnStop.bValue				:= TRUE;

			tyP1031MagSetTeach.tyTeachLifterMag4Slt1Pos.tyBtn2.bRtLk			:= FALSE;
			tyP1031MagSetTeach.tyMotionStdLifter.tyBtnStop.bRtLk				:= TRUE;
		END_IF

	ELSIF tyP1031MagSetTeach.tyMotionStdLifter.tyBtnMovAbs.bRtCompl = TRUE THEN

		tyP1031MagSetTeach.tyMotionStdLifter.tyBtnMovAbs.bValue				:= TRUE;
		tyP1031MagSetTeach.tyMotionStdLifter.tyBtnStop.bValue				:= FALSE;

		tyP1031MagSetTeach.tyMotionStdLifter.tyBtnMovAbs.bRtLk				:= TRUE;
		tyP1031MagSetTeach.tyMotionStdLifter.tyBtnStop.bRtLk					:= FALSE;

		diMnlLifterTargetPos	:= tyP1031MagSetTeach.tyMotionStdLifter.tyNumTargetPos.diValue;
		diMnlLifterNomSpd		:= tyP1031MagSetTeach.tyMotionStdLifter.tyNumNomSpd.diValue;

		eLifterBtmAct			:= LifterActMovAbs;

		IF p_eLifterBtmStat = LifterActMovAbs AND p_eLifterBtmStatus = Done THEN
			eLifterBtmAct	:= LifterActIdle;

			tyP1031MagSetTeach.tyMotionStdLifter.tyBtnMovAbs.bRtCompl	:= FALSE;
			tyP1031MagSetTeach.tyMotionStdLifter.tyBtnMovAbs.bValue		:= FALSE;
			tyP1031MagSetTeach.tyMotionStdLifter.tyBtnStop.bValue		:= TRUE;

			tyP1031MagSetTeach.tyMotionStdLifter.tyBtnMovAbs.bRtLk		:= FALSE;
			tyP1031MagSetTeach.tyMotionStdLifter.tyBtnStop.bRtLk		:= TRUE;
		END_IF

	ELSIF tyP1031MagSetTeach.tyMotionStdLifter.tyBtnMovRel.bRtCompl = TRUE THEN
		tyP1031MagSetTeach.tyMotionStdLifter.tyBtnMovRel.bValue			:= TRUE;
		tyP1031MagSetTeach.tyMotionStdLifter.tyBtnStop.bValue			:= FALSE;

		tyP1031MagSetTeach.tyMotionStdLifter.tyBtnMovRel.bRtLk			:= TRUE;
		tyP1031MagSetTeach.tyMotionStdLifter.tyBtnStop.bRtLk				:= FALSE;

		diMnlLifterStepSize		:= tyP1031MagSetTeach.tyMotionStdLifter.tyNumStepSize.diValue;
		diMnlLifterNomSpd		:= tyP1031MagSetTeach.tyMotionStdLifter.tyNumNomSpd.diValue;

		eLifterBtmAct		:= LifterActMovRel;

		IF p_eLifterBtmStat = LifterActMovRel AND p_eLifterBtmStatus = Done THEN
			eLifterBtmAct	:= LifterActIdle;

			tyP1031MagSetTeach.tyMotionStdLifter.tyBtnMovRel.bRtCompl		:= FALSE;
			tyP1031MagSetTeach.tyMotionStdLifter.tyBtnMovRel.bValue			:= FALSE;
			tyP1031MagSetTeach.tyMotionStdLifter.tyBtnStop.bValue			:= TRUE;

			tyP1031MagSetTeach.tyMotionStdLifter.tyBtnMovRel.bRtLk			:= FALSE;
			tyP1031MagSetTeach.tyMotionStdLifter.tyBtnStop.bRtLk				:= TRUE;

		END_IF

	ELSIF (tyP1031MagSetTeach.tyMotionStdLifter.tyBtnJogDown.bValue = TRUE) AND (fbJogSlowToFastDlyTm.Q = FALSE) AND (bJogSlow = FALSE) THEN
		tyP1031MagSetTeach.tyMotionStdLifter.tyBtnStop.bValue				:= FALSE;
		tyP1031MagSetTeach.tyMotionStdLifter.tyBtnStop.bRtLk				:= FALSE;

		fbJogSlowToFastDlyTm.IN		:= TRUE;

		diMnlLifterJogSpd	:= tyP1031MagSetTeach.tyMotionStdLifter.tyNumSlwSpd.diValue;

		eLifterBtmAct		:= LifterActJogDown;

		IF p_eLifterBtmStat = LifterActJogDown AND p_eLifterBtmStatus = Done THEN

			eLifterBtmAct	:= LifterActIdle;
			bJogSlow				:= TRUE;

		ELSIF p_eLifterBtmStatus = Error THEN

			fbJogSlowToFastDlyTm.IN	:= FALSE;
			bJogSlow				:= TRUE;

		END_IF

	ELSIF (tyP1031MagSetTeach.tyMotionStdLifter.tyBtnJogDown.bValue = TRUE) AND (fbJogSlowToFastDlyTm.Q = TRUE) AND (bJogFast = FALSE) THEN
		tyP1031MagSetTeach.tyMotionStdLifter.tyBtnStop.bValue					:= FALSE;
		tyP1031MagSetTeach.tyMotionStdLifter.tyBtnStop.bRtLk					:= FALSE;

		fbJogSlowToFastDlyTm.IN		:= TRUE;

		diMnlLifterJogSpd	:= tyP1031MagSetTeach.tyMotionStdLifter.tyNumNomSpd.diValue;

		eLifterBtmAct		:= LifterActJogDown;

		IF p_eLifterBtmStat = LifterActJogDown AND p_eLifterBtmStatus = Done THEN
			eLifterBtmAct	:= LifterActIdle;
			bJogFast				:= TRUE;
		ELSIF p_eLifterBtmStatus = Error THEN
			fbJogSlowToFastDlyTm.IN	:= FALSE;
			bJogFast				:= TRUE;
		END_IF

	ELSIF (tyP1031MagSetTeach.tyMotionStdLifter.tyBtnJogUp.bValue = TRUE) AND (fbJogSlowToFastDlyTm.Q = FALSE) AND (bJogSlow = FALSE) THEN
		tyP1031MagSetTeach.tyMotionStdLifter.tyBtnStop.bValue				:= FALSE;
		tyP1031MagSetTeach.tyMotionStdLifter.tyBtnStop.bRtLk				:= FALSE;

		fbJogSlowToFastDlyTm.IN		:= TRUE;

		diMnlLifterJogSpd	:= tyP1031MagSetTeach.tyMotionStdLifter.tyNumSlwSpd.diValue;

		eLifterBtmAct		:= LifterActJogUp;

		IF p_eLifterBtmStat = LifterActJogUp AND p_eLifterBtmStatus = Done THEN
			eLifterBtmAct	:= LifterActIdle;
			bJogSlow				:= TRUE;

		ELSIF p_eLifterBtmStatus = Error THEN
			fbJogSlowToFastDlyTm.IN	:= FALSE;
			bJogSlow				:= TRUE;
		END_IF

	ELSIF (tyP1031MagSetTeach.tyMotionStdLifter.tyBtnJogUp.bValue = TRUE) AND (fbJogSlowToFastDlyTm.Q = TRUE) AND (bJogFast = FALSE) THEN

		tyP1031MagSetTeach.tyMotionStdLifter.tyBtnStop.bValue				:= FALSE;
		tyP1031MagSetTeach.tyMotionStdLifter.tyBtnStop.bRtLk					:= FALSE;

		fbJogSlowToFastDlyTm.IN		:= TRUE;

		diMnlLifterJogSpd	:= tyP1031MagSetTeach.tyMotionStdLifter.tyNumNomSpd.diValue;

		eLifterBtmAct		:= LifterActJogUp;

		IF p_eLifterBtmStat = LifterActJogUp AND p_eLifterBtmStatus = Done THEN
			eLifterBtmAct	:= LifterActIdle;
			bJogFast	:= TRUE;

		ELSIF p_eLifterBtmStatus = Error THEN
			fbJogSlowToFastDlyTm.IN	:= FALSE;
			bJogFast				:= TRUE;
		END_IF
	END_IF

	IF tyP1031MagSetTeach.tyInOutletShutterFB.tyBtnOpen.bRtCompl = TRUE THEN
		tyP1031MagSetTeach.tyInOutletShutterFB.tyBtnOpen.bRtCompl	:= FALSE;

		tyP1031MagSetTeach.tyInOutletShutterFB.tyBtnOpen.bValue	:= TRUE;
		tyP1031MagSetTeach.tyInOutletShutterFB.tyBtnClose.bValue	:= FALSE;

	ELSIF tyP1031MagSetTeach.tyInOutletShutterFB.tyBtnClose.bRtCompl = TRUE THEN
		tyP1031MagSetTeach.tyInOutletShutterFB.tyBtnClose.bRtCompl	:= FALSE;

		tyP1031MagSetTeach.tyInOutletShutterFB.tyBtnClose.bValue	:= TRUE;
		tyP1031MagSetTeach.tyInOutletShutterFB.tyBtnOpen.bValue	:= FALSE;
	END_IF

	IF tyP1031MagSetTeach.tyInOutletShutterFB.tyBtnOpen.bValue = TRUE THEN
		eInShutterAct	:= PneuActRet;
		eOutShutterAct	:= PneuActRet;

		IF (p_eInShutterStat = PneuActRet AND p_eInShutterStatus = Done)
			AND (p_eOutShutterStat = PneuActRet AND p_eOutShutterStatus = Done)
			THEN
			eInShutterAct	:= PneuActIdle;
			eOutShutterAct	:= PneuActIdle;
			tyP1031MagSetTeach.tyInOutletShutterFB.tyBtnOpen.bValue	:= FALSE;
		ELSIF p_eInShutterStatus = Error OR p_eOutShutterStatus = Error THEN
			tyP1031MagSetTeach.tyInOutletShutterFB.tyBtnOpen.bValue	:= FALSE;
		END_IF

	ELSIF tyP1031MagSetTeach.tyInOutletShutterFB.tyBtnClose.bValue = TRUE THEN
		eInShutterAct	:= PneuActExt;
		eOutShutterAct	:= PneuActExt;
		IF (p_eInShutterStat = PneuActExt AND p_eInShutterStatus = Done)
			AND (p_eOutShutterStat = PneuActExt AND p_eOutShutterStatus = Done)
			THEN
			eInShutterAct	:= PneuActIdle;
			eOutShutterAct	:= PneuActIdle;
			tyP1031MagSetTeach.tyInOutletShutterFB.tyBtnClose.bValue := FALSE;
		ELSIF p_eInShutterStatus = Error OR p_eOutShutterStatus = Error THEN
			tyP1031MagSetTeach.tyInOutletShutterFB.tyBtnClose.bValue := FALSE;
		END_IF
	END_IF

	//bypass curtain sensor
	IF bTeachLifterMag1Slt1Pos OR bTeachLifterMag2Slt1Pos OR bTeachLifterMag3Slt1Pos THEN
		bBypCurtainSen			:= tyP1031MagSetTeach.tyTeachLifterMag1Slt1Pos.tyBtn4.bValue OR tyP1031MagSetTeach.tyTeachLifterMag2Slt1Pos.tyBtn4.bValue OR tyP1031MagSetTeach.tyTeachLifterMag3Slt1Pos.tyBtn4.bValue;
		bBypCurtainPBLED		:= tyP1031MagSetTeach.tyTeachLifterMag1Slt1Pos.tyBtn4.bValue OR tyP1031MagSetTeach.tyTeachLifterMag2Slt1Pos.tyBtn4.bValue OR tyP1031MagSetTeach.tyTeachLifterMag3Slt1Pos.tyBtn4.bValue;
	END_IF

END_ACTION
```
